LIN {X 0,Y 457.677,Z 380.613,A -85,B 0,C 180,E1 -16942.312,E2 -16942.312} C_VEL
LIN {X 0,Y 452.444,Z 370.143,A -85,B 0,C 180,E1 -16943.24,E2 -16943.24} C_VEL
LIN {X 0,Y 446.614,Z 360.173,A -85,B 0,C 180,E1 -16944.308,E2 -16944.308} C_VEL
LIN {X 0,Y 441.723,Z 352.476,A -85,B 0,C 180,E1 -16945.27,E2 -16945.27} C_VEL
LIN {X 0,Y 439.765,Z 349.442,A -85,B 0,C 180,E1 -16945.668,E2 -16945.668} C_VEL
LIN {X 0,Y 438.909,Z 348.163,A -85,B 0,C 180,E1 -16945.842,E2 -16945.842} C_VEL
LIN {X 0,Y 436.998,Z 345.517,A -85,B 0,C 180,E1 -16946.247,E2 -16946.247} C_VEL
LIN {X 0,Y 436.487,Z 343.674,A -85,B 0,C 180,E1 -16946.435,E2 -16946.435} C_VEL
LIN {X 0,Y 436.475,Z 343.673,A -85,B 0,C 180,E1 -16948.779,E2 -16948.779} C_VEL
LIN {X 0,Y 436.468,Z 343.672,A -85,B 0,C 180,E1 -16951.977,E2 -16951.977} C_VEL
LIN {X 0,Y 436.477,Z 343.666,A -85,B 0,C 180,E1 -16955.29,E2 -16955.29} C_VEL
LIN {X 0,Y 436.436,Z 343.668,A -85,B 0,C 180,E1 -16958.75,E2 -16958.75} C_VEL
LIN {X 0,Y 436.445,Z 343.67,A -85,B 0,C 180,E1 -16961.148,E2 -16961.148} C_VEL
LIN {X 0,Y 436.447,Z 343.671,A -85,B 0,C 180,E1 -16963.764,E2 -16963.764} C_VEL
LIN {X 0,Y 436.45,Z 343.673,A -85,B 0,C 180,E1 -16966.362,E2 -16966.362} C_VEL
LIN {X 0,Y 436.423,Z 343.682,A -85,B 0,C 180,E1 -16968.967,E2 -16968.967} C_VEL
LIN {X 0,Y 436.425,Z 343.682,A -85,B 0,C 180,E1 -16972.419,E2 -16972.419} C_VEL
LIN {X 0,Y 436.431,Z 343.811,A -85,B 0,C 180,E1 -16975.755,E2 -16975.755} C_VEL
LIN {X 0,Y 440.459,Z 359.383,A -85,B 0,C 180,E1 -16978.559,E2 -16978.559} C_VEL
LIN {X 0,Y 443.529,Z 373.428,A -85,B 0,C 180,E1 -16980.947,E2 -16980.947} C_VEL
LIN {X 0,Y 444.042,Z 376.825,A -85,B 0,C 180,E1 -16981.499,E2 -16981.499} C_VEL
LIN {X 0,Y 442.672,Z 390.65,A -85,B 0,C 180,E1 -16983.511,E2 -16983.511} C_VEL
LIN {X 0,Y 443.709,Z 396.754,A -85,B 0,C 180,E1 -16983.869,E2 -16983.869} C_VEL
LIN {X 0,Y 447.375,Z 420.193,A -85,B 0,C 180,E1 -16985.137,E2 -16985.137} C_VEL
LIN {X 0,Y 449.599,Z 437.106,A -85,B 0,C 180,E1 -16985.947,E2 -16985.947} C_VEL
LIN {X 0,Y 451.261,Z 453.177,A -85,B 0,C 180,E1 -16986.628,E2 -16986.628} C_VEL
LIN {X 0,Y 452.377,Z 476.599,A -85,B 0,C 180,E1 -16987.477,E2 -16987.477} C_VEL
LIN {X 0,Y 448.009,Z 553.44,A -85,B 0,C 180,E1 -16989.404,E2 -16989.404} C_VEL
LIN {X 0,Y 446.573,Z 569.624,A -85,B 0,C 180,E1 -16989.993,E2 -16989.993} C_VEL
LIN {X 0,Y 444.876,Z 583.938,A -85,B 0,C 180,E1 -16990.692,E2 -16990.692} C_VEL
LIN {X 0,Y 443.084,Z 597.736,A -85,B 0,C 180,E1 -16991.568,E2 -16991.568} C_VEL
LIN {X 0,Y 440.902,Z 615.075,A -85,B 0,C 180,E1 -16992.908,E2 -16992.908} C_VEL
LIN {X 0,Y 439.422,Z 626.686,A -85,B 0,C 180,E1 -16994.04,E2 -16994.04} C_VEL
LIN {X 0,Y 438.078,Z 636.36,A -85,B 0,C 180,E1 -16995.177,E2 -16995.177} C_VEL
LIN {X 0,Y 436.955,Z 646.109,A -85,B 0,C 180,E1 -16996.559,E2 -16996.559} C_VEL
LIN {X 0,Y 436.4,Z 651.742,A -85,B 0,C 180,E1 -16997.486,E2 -16997.486} C_VEL
LIN {X 0,Y 435.744,Z 662.573,A -85,B 0,C 180,E1 -16998.749,E2 -16998.749} C_VEL
LIN {X 0,Y 435.303,Z 671.76,A -85,B 0,C 180,E1 -17000.039,E2 -17000.039} C_VEL
LIN {X 0,Y 434.928,Z 680.021,A -85,B 0,C 180,E1 -17001.433,E2 -17001.433} C_VEL
LIN {X 0,Y 434.668,Z 687.893,A -85,B 0,C 180,E1 -17003.058,E2 -17003.058} C_VEL
LIN {X 0,Y 434.564,Z 693.312,A -85,B 0,C 180,E1 -17004.45,E2 -17004.45} C_VEL
LIN {X 0,Y 434.439,Z 697.641,A -85,B 0,C 180,E1 -17005.839,E2 -17005.839} C_VEL
LIN {X 0,Y 434.396,Z 701.016,A -85,B 0,C 180,E1 -17007.227,E2 -17007.227} C_VEL
LIN {X 0,Y 434.402,Z 703.511,A -85,B 0,C 180,E1 -17008.614,E2 -17008.614} C_VEL
LIN {X 0,Y 434.384,Z 705.081,A -85,B 0,C 180,E1 -17010,E2 -17010} C_VEL
LIN {X 0,Y 434.419,Z 705.916,A -85,B 0,C 180,E1 -17011.848,E2 -17011.848} C_VEL
LIN {X 0,Y 434.466,Z 705.265,A -85,B 0,C 180,E1 -17013.697,E2 -17013.697} C_VEL
LIN {X 0,Y 434.713,Z 703.119,A -85,B 0,C 180,E1 -17015.548,E2 -17015.548} C_VEL
LIN {X 0,Y 435.174,Z 699.48,A -85,B 0,C 180,E1 -17017.398,E2 -17017.398} C_VEL
LIN {X 0,Y 435.868,Z 694.257,A -85,B 0,C 180,E1 -17019.247,E2 -17019.247} C_VEL
LIN {X 0,Y 436.699,Z 689.192,A -85,B 0,C 180,E1 -17020.629,E2 -17020.629} C_VEL
LIN {X 0,Y 437.941,Z 681.532,A -85,B 0,C 180,E1 -17022.309,E2 -17022.309} C_VEL
LIN {X 0,Y 439.27,Z 672.935,A -85,B 0,C 180,E1 -17023.838,E2 -17023.838} C_VEL
LIN {X 0,Y 440.847,Z 663.536,A -85,B 0,C 180,E1 -17025.198,E2 -17025.198} C_VEL
LIN {X 0,Y 442.451,Z 652.225,A -85,B 0,C 180,E1 -17026.556,E2 -17026.556} C_VEL
LIN {X 0,Y 444.327,Z 639.573,A -85,B 0,C 180,E1 -17027.784,E2 -17027.784} C_VEL
LIN {X 0,Y 446.052,Z 626.94,A -85,B 0,C 180,E1 -17028.779,E2 -17028.779} C_VEL
LIN {X 0,Y 447.529,Z 613.948,A -85,B 0,C 180,E1 -17029.604,E2 -17029.604} C_VEL
LIN {X 0,Y 449.037,Z 599.167,A -85,B 0,C 180,E1 -17030.328,E2 -17030.328} C_VEL
LIN {X 0,Y 450.408,Z 583.991,A -85,B 0,C 180,E1 -17030.866,E2 -17030.866} C_VEL
LIN {X 0,Y 456.645,Z 487.44,A -85,B 0,C 180,E1 -17033.354,E2 -17033.354} C_VEL
LIN {X 0,Y 457.242,Z 476.209,A -85,B 0,C 180,E1 -17033.674,E2 -17033.674} C_VEL
LIN {X 0,Y 456.643,Z 460.353,A -85,B 0,C 180,E1 -17034.284,E2 -17034.284} C_VEL
LIN {X 0,Y 454.633,Z 438.662,A -85,B 0,C 180,E1 -17035.296,E2 -17035.296} C_VEL
LIN {X 0,Y 454.42,Z 436.088,A -85,B 0,C 180,E1 -17035.446,E2 -17035.446} C_VEL
LIN {X 0,Y 454.349,Z 415.095,A -85,B 0,C 180,E1 -17037.094,E2 -17037.094} C_VEL
LIN {X 0,Y 454.414,Z 399.172,A -85,B 0,C 180,E1 -17038.545,E2 -17038.545} C_VEL
LIN {X 0,Y 454.669,Z 389.171,A -85,B 0,C 180,E1 -17039.537,E2 -17039.537} C_VEL
LIN {X 0,Y 454.757,Z 385.084,A -85,B 0,C 180,E1 -17039.972,E2 -17039.972} C_VEL
LIN {X 0,Y 453.574,Z 375.492,A -85,B 0,C 180,E1 -17041.419,E2 -17041.419} C_VEL
LIN {X 0,Y 453.221,Z 371.903,A -85,B 0,C 180,E1 -17042.027,E2 -17042.027} C_VEL
LIN {X 0,Y 451.396,Z 368.316,A -85,B 0,C 180,E1 -17043.078,E2 -17043.078} C_VEL
LIN {X 0,Y 448.758,Z 363.877,A -85,B 0,C 180,E1 -17044.765,E2 -17044.765} C_VEL
LIN {X 0,Y 446.279,Z 359.984,A -85,B 0,C 180,E1 -17046.826,E2 -17046.826} C_VEL
LIN {X 0,Y 445.144,Z 358.305,A -85,B 0,C 180,E1 -17048.116,E2 -17048.116} C_VEL
LIN {X 0,Y 443.873,Z 356.858,A -85,B 0,C 180,E1 -17050.315,E2 -17050.315} C_VEL
LIN {X 0,Y 443.562,Z 356.547,A -85,B 0,C 180,E1 -17052.082,E2 -17052.082} C_VEL
LIN {X 0,Y 443.886,Z 357.081,A -85,B 0,C 180,E1 -17053.972,E2 -17053.972} C_VEL
LIN {X 0,Y 444.508,Z 357.779,A -85,B 0,C 180,E1 -17055.162,E2 -17055.162} C_VEL
LIN {X 0,Y 445.079,Z 359.312,A -85,B 0,C 180,E1 -17056.38,E2 -17056.38} C_VEL
LIN {X 0,Y 446.306,Z 361.926,A -85,B 0,C 180,E1 -17058.075,E2 -17058.075} C_VEL
LIN {X 0,Y 448.189,Z 366.353,A -85,B 0,C 180,E1 -17060.152,E2 -17060.152} C_VEL
LIN {X 0,Y 450.674,Z 372.66,A -85,B 0,C 180,E1 -17062.434,E2 -17062.434} C_VEL
LIN {X 0,Y 452.888,Z 379.057,A -85,B 0,C 180,E1 -17064.318,E2 -17064.318} C_VEL
LIN {X 0,Y 455.207,Z 387.381,A -85,B 0,C 180,E1 -17066.362,E2 -17066.362} C_VEL
LIN {X 0,Y 457.231,Z 396.879,A -85,B 0,C 180,E1 -17068.361,E2 -17068.361} C_VEL
LIN {X 0,Y 457.648,Z 400.955,A -85,B 0,C 180,E1 -17069.093,E2 -17069.093} C_VEL
LIN {X 0,Y 454.383,Z 422.257,A -85,B 0,C 180,E1 -17072.001,E2 -17072.001} C_VEL
LIN {X 0,Y 451.946,Z 440.08,A -85,B 0,C 180,E1 -17074.351,E2 -17074.351} C_VEL
LIN {X 0,Y 455.098,Z 456.713,A -85,B 0,C 180,E1 -17075.326,E2 -17075.326} C_VEL
LIN {X 0,Y 457.268,Z 472.318,A -85,B 0,C 180,E1 -17076.103,E2 -17076.103} C_VEL
LIN {X 0,Y 457.699,Z 477.669,A -85,B 0,C 180,E1 -17076.329,E2 -17076.329} C_VEL
LIN {X 0,Y 452.325,Z 559.762,A -85,B 0,C 180,E1 -17078.428,E2 -17078.428} C_VEL
LIN {X 0,Y 450.776,Z 583.934,A -85,B 0,C 180,E1 -17079.06,E2 -17079.06} C_VEL
LIN {X 0,Y 449.354,Z 599.265,A -85,B 0,C 180,E1 -17079.647,E2 -17079.647} C_VEL
LIN {X 0,Y 447.901,Z 613.022,A -85,B 0,C 180,E1 -17080.353,E2 -17080.353} C_VEL
LIN {X 0,Y 446.285,Z 626.426,A -85,B 0,C 180,E1 -17081.232,E2 -17081.232} C_VEL
LIN {X 0,Y 444.402,Z 639.894,A -85,B 0,C 180,E1 -17082.338,E2 -17082.338} C_VEL
LIN {X 0,Y 442.623,Z 652.052,A -85,B 0,C 180,E1 -17083.569,E2 -17083.569} C_VEL
LIN {X 0,Y 440.999,Z 662.166,A -85,B 0,C 180,E1 -17084.807,E2 -17084.807} C_VEL
LIN {X 0,Y 439.496,Z 671.417,A -85,B 0,C 180,E1 -17086.169,E2 -17086.169} C_VEL
LIN {X 0,Y 438.119,Z 680.312,A -85,B 0,C 180,E1 -17087.782,E2 -17087.782} C_VEL
LIN {X 0,Y 436.881,Z 687.469,A -85,B 0,C 180,E1 -17089.375,E2 -17089.375} C_VEL
LIN {X 0,Y 436.048,Z 692.49,A -85,B 0,C 180,E1 -17090.756,E2 -17090.756} C_VEL
LIN {X 0,Y 435.249,Z 697.663,A -85,B 0,C 180,E1 -17092.603,E2 -17092.603} C_VEL
LIN {X 0,Y 434.706,Z 701.272,A -85,B 0,C 180,E1 -17094.452,E2 -17094.452} C_VEL
LIN {X 0,Y 434.444,Z 703.403,A -85,B 0,C 180,E1 -17096.303,E2 -17096.303} C_VEL
LIN {X 0,Y 434.35,Z 704.067,A -85,B 0,C 180,E1 -17098.152,E2 -17098.152} C_VEL
LIN {X 0,Y 434.316,Z 703.251,A -85,B 0,C 180,E1 -17100,E2 -17100} C_VEL
LIN {X 0,Y 434.35,Z 700.967,A -85,B 0,C 180,E1 -17101.849,E2 -17101.849} C_VEL
LIN {X 0,Y 434.349,Z 698.27,A -85,B 0,C 180,E1 -17103.236,E2 -17103.236} C_VEL
LIN {X 0,Y 434.441,Z 694.648,A -85,B 0,C 180,E1 -17104.624,E2 -17104.624} C_VEL
LIN {X 0,Y 434.575,Z 689.804,A -85,B 0,C 180,E1 -17106.07,E2 -17106.07} C_VEL
LIN {X 0,Y 434.826,Z 683.278,A -85,B 0,C 180,E1 -17107.637,E2 -17107.637} C_VEL
LIN {X 0,Y 435.223,Z 674.843,A -85,B 0,C 180,E1 -17109.262,E2 -17109.262} C_VEL
LIN {X 0,Y 435.755,Z 665.995,A -85,B 0,C 180,E1 -17110.653,E2 -17110.653} C_VEL
LIN {X 0,Y 436.232,Z 656.984,A -85,B 0,C 180,E1 -17111.843,E2 -17111.843} C_VEL
LIN {X 0,Y 436.876,Z 645.666,A -85,B 0,C 180,E1 -17113.089,E2 -17113.089} C_VEL
LIN {X 0,Y 437.653,Z 632.877,A -85,B 0,C 180,E1 -17114.245,E2 -17114.245} C_VEL
LIN {X 0,Y 438.37,Z 620.317,A -85,B 0,C 180,E1 -17115.168,E2 -17115.168} C_VEL
LIN {X 0,Y 439.097,Z 606.466,A -85,B 0,C 180,E1 -17115.973,E2 -17115.973} C_VEL
LIN {X 0,Y 439.608,Z 592.172,A -85,B 0,C 180,E1 -17116.607,E2 -17116.607} C_VEL
LIN {X 0,Y 440.169,Z 576.613,A -85,B 0,C 180,E1 -17117.094,E2 -17117.094} C_VEL
LIN {X 0,Y 442.754,Z 469.934,A -85,B 0,C 180,E1 -17119.451,E2 -17119.451} C_VEL
LIN {X 0,Y 439.834,Z 439.603,A -85,B 0,C 180,E1 -17120.233,E2 -17120.233} C_VEL
LIN {X 0,Y 441.544,Z 410.298,A -85,B 0,C 180,E1 -17123.861,E2 -17123.861} C_VEL
LIN {X 0,Y 443.123,Z 384.772,A -85,B 0,C 180,E1 -17127.03,E2 -17127.03} C_VEL
LIN {X 0,Y 443.661,Z 375.927,A -85,B 0,C 180,E1 -17128.132,E2 -17128.132} C_VEL
LIN {X 0,Y 439.991,Z 358.902,A -85,B 0,C 180,E1 -17130.454,E2 -17130.454} C_VEL
LIN {X 0,Y 436.523,Z 343.668,A -85,B 0,C 180,E1 -17132.584,E2 -17132.584} C_VEL
LIN {X 0,Y 436.491,Z 343.675,A -85,B 0,C 180,E1 -17135.289,E2 -17135.289} C_VEL
LIN {X 0,Y 436.468,Z 343.673,A -85,B 0,C 180,E1 -17138.747,E2 -17138.747} C_VEL
LIN {X 0,Y 436.48,Z 343.675,A -85,B 0,C 180,E1 -17141.144,E2 -17141.144} C_VEL
LIN {X 0,Y 436.472,Z 343.67,A -85,B 0,C 180,E1 -17143.767,E2 -17143.767} C_VEL
LIN {X 0,Y 436.472,Z 343.671,A -85,B 0,C 180,E1 -17146.365,E2 -17146.365} C_VEL
LIN {X 0,Y 436.483,Z 343.674,A -85,B 0,C 180,E1 -17148.959,E2 -17148.959} C_VEL
LIN {X 0,Y 436.459,Z 343.675,A -85,B 0,C 180,E1 -17152.422,E2 -17152.422} C_VEL
LIN {X 0,Y 436.479,Z 343.669,A -85,B 0,C 180,E1 -17155.829,E2 -17155.829} C_VEL
LIN {X 0,Y 436.467,Z 343.671,A -85,B 0,C 180,E1 -17159.1,E2 -17159.1} C_VEL
LIN {X 0,Y 436.5,Z 343.672,A -85,B 0,C 180,E1 -17162.267,E2 -17162.267} C_VEL
LIN {X 0,Y 436.453,Z 343.672,A -85,B 0,C 180,E1 -17165.338,E2 -17165.338} C_VEL
LIN {X 0,Y 436.49,Z 343.674,A -85,B 0,C 180,E1 -17168.341,E2 -17168.341} C_VEL
LIN {X 0,Y 436.536,Z 343.663,A -85,B 0,C 180,E1 -17171.282,E2 -17171.282} C_VEL
LIN {X 0,Y 436.539,Z 343.669,A -85,B 0,C 180,E1 -17173.973,E2 -17173.973} C_VEL
LIN {X 0,Y 438.742,Z 349.624,A -85,B 0,C 180,E1 -17174.188,E2 -17174.188} C_VEL
LIN {X 0,Y 445.557,Z 367.49,A -85,B 0,C 180,E1 -17174.799,E2 -17174.799} C_VEL
LIN {X 0,Y 444.443,Z 456.819,A -85,B 0,C 180,E1 -17176.24,E2 -17176.24} C_VEL
LIN {X 0,Y 444.336,Z 471.415,A -85,B 0,C 180,E1 -17176.584,E2 -17176.584} C_VEL
LIN {X 0,Y 443.999,Z 484.727,A -85,B 0,C 180,E1 -17177.067,E2 -17177.067} C_VEL
LIN {X 0,Y 443.418,Z 497.369,A -85,B 0,C 180,E1 -17177.687,E2 -17177.687} C_VEL
LIN {X 0,Y 442.709,Z 509.826,A -85,B 0,C 180,E1 -17178.478,E2 -17178.478} C_VEL
LIN {X 0,Y 441.998,Z 522.081,A -85,B 0,C 180,E1 -17179.46,E2 -17179.46} C_VEL
LIN {X 0,Y 440.993,Z 533.977,A -85,B 0,C 180,E1 -17180.63,E2 -17180.63} C_VEL
LIN {X 0,Y 440.059,Z 543.484,A -85,B 0,C 180,E1 -17181.764,E2 -17181.764} C_VEL
LIN {X 0,Y 439.03,Z 553.01,A -85,B 0,C 180,E1 -17183.128,E2 -17183.128} C_VEL
LIN {X 0,Y 438.195,Z 560.908,A -85,B 0,C 180,E1 -17184.497,E2 -17184.497} C_VEL
LIN {X 0,Y 437.468,Z 567.499,A -85,B 0,C 180,E1 -17185.868,E2 -17185.868} C_VEL
LIN {X 0,Y 436.897,Z 572.99,A -85,B 0,C 180,E1 -17187.243,E2 -17187.243} C_VEL
LIN {X 0,Y 436.368,Z 578.741,A -85,B 0,C 180,E1 -17189.08,E2 -17189.08} C_VEL
LIN {X 0,Y 436.014,Z 582.966,A -85,B 0,C 180,E1 -17190.921,E2 -17190.921} C_VEL
LIN {X 0,Y 435.921,Z 585.784,A -85,B 0,C 180,E1 -17192.763,E2 -17192.763} C_VEL
LIN {X 0,Y 435.817,Z 587.301,A -85,B 0,C 180,E1 -17194.609,E2 -17194.609} C_VEL
LIN {X 0,Y 436.001,Z 587.512,A -85,B 0,C 180,E1 -17196.457,E2 -17196.457} C_VEL
LIN {X 0,Y 436.222,Z 586.445,A -85,B 0,C 180,E1 -17198.309,E2 -17198.309} C_VEL
LIN {X 0,Y 436.612,Z 584.058,A -85,B 0,C 180,E1 -17200.164,E2 -17200.164} C_VEL
LIN {X 0,Y 437.413,Z 580.231,A -85,B 0,C 180,E1 -17202.016,E2 -17202.016} C_VEL
LIN {X 0,Y 438.269,Z 574.861,A -85,B 0,C 180,E1 -17203.871,E2 -17203.871} C_VEL
LIN {X 0,Y 439.123,Z 569.75,A -85,B 0,C 180,E1 -17205.26,E2 -17205.26} C_VEL
LIN {X 0,Y 440.079,Z 563.506,A -85,B 0,C 180,E1 -17206.648,E2 -17206.648} C_VEL
LIN {X 0,Y 440.565,Z 560.276,A -85,B 0,C 180,E1 -17207.273,E2 -17207.273} C_VEL
LIN {X 0,Y 440.422,Z 556.973,A -85,B 0,C 180,E1 -17207.912,E2 -17207.912} C_VEL
LIN {X 0,Y 438.511,Z 551.47,A -85,B 0,C 180,E1 -17208.962,E2 -17208.962} C_VEL
LIN {X 0,Y 436.643,Z 545.441,A -85,B 0,C 180,E1 -17209.963,E2 -17209.963} C_VEL
LIN {X 0,Y 436.555,Z 541.317,A -85,B 0,C 180,E1 -17210.517,E2 -17210.517} C_VEL
LIN {X 0,Y 437.884,Z 530.282,A -85,B 0,C 180,E1 -17211.755,E2 -17211.755} C_VEL
LIN {X 0,Y 439.035,Z 519.376,A -85,B 0,C 180,E1 -17212.761,E2 -17212.761} C_VEL
LIN {X 0,Y 440.224,Z 506.915,A -85,B 0,C 180,E1 -17213.688,E2 -17213.688} C_VEL
LIN {X 0,Y 440.86,Z 495.16,A -85,B 0,C 180,E1 -17214.399,E2 -17214.399} C_VEL
LIN {X 0,Y 441.544,Z 480.938,A -85,B 0,C 180,E1 -17215.046,E2 -17215.046} C_VEL
LIN {X 0,Y 441.906,Z 467.059,A -85,B 0,C 180,E1 -17215.486,E2 -17215.486} C_VEL
LIN {X 0,Y 442.223,Z 442.075,A -85,B 0,C 180,E1 -17215.945,E2 -17215.945} C_VEL
LIN {X 0,Y 443.528,Z 375.813,A -85,B 0,C 180,E1 -17217.024,E2 -17217.024} C_VEL
LIN {X 0,Y 433.277,Z 353.124,A -85,B 0,C 180,E1 -17218.061,E2 -17218.061} C_VEL
LIN {X 0,Y 429.628,Z 345.62,A -85,B 0,C 180,E1 -17218.434,E2 -17218.434} C_VEL
LIN {X 0,Y 429.415,Z 344.551,A -85,B 0,C 180,E1 -17218.479,E2 -17218.479} C_VEL
LIN {X 0,Y 429.376,Z 344.556,A -85,B 0,C 180,E1 -17221.468,E2 -17221.468} C_VEL
LIN {X 0,Y 429.34,Z 344.563,A -85,B 0,C 180,E1 -17224.821,E2 -17224.821} C_VEL
LIN {X 0,Y 429.386,Z 344.556,A -85,B 0,C 180,E1 -17227.126,E2 -17227.126} C_VEL
LIN {X 0,Y 429.37,Z 344.561,A -85,B 0,C 180,E1 -17230.733,E2 -17230.733} C_VEL
LIN {X 0,Y 429.394,Z 344.557,A -85,B 0,C 180,E1 -17234.131,E2 -17234.131} C_VEL
LIN {X 0,Y 429.383,Z 344.556,A -85,B 0,C 180,E1 -17237.23,E2 -17237.23} C_VEL
LIN {X 0,Y 429.369,Z 344.553,A -85,B 0,C 180,E1 -17240.489,E2 -17240.489} C_VEL
LIN {X 0,Y 429.383,Z 344.521,A -85,B 0,C 180,E1 -17243.066,E2 -17243.066} C_VEL
LIN {X 0,Y 429.393,Z 344.553,A -85,B 0,C 180,E1 -17246.315,E2 -17246.315} C_VEL
LIN {X 0,Y 429.408,Z 344.545,A -85,B 0,C 180,E1 -17249.83,E2 -17249.83} C_VEL
LIN {X 0,Y 429.427,Z 344.546,A -85,B 0,C 180,E1 -17252.824,E2 -17252.824} C_VEL
LIN {X 0,Y 429.42,Z 344.554,A -85,B 0,C 180,E1 -17255.986,E2 -17255.986} C_VEL
LIN {X 0,Y 429.446,Z 344.543,A -85,B 0,C 180,E1 -17259.386,E2 -17259.386} C_VEL
LIN {X 0,Y 435.371,Z 365.507,A -85,B 0,C 180,E1 -17260.041,E2 -17260.041} C_VEL
LIN {X 0,Y 433.262,Z 463.185,A -85,B 0,C 180,E1 -17262.23,E2 -17262.23} C_VEL
LIN {X 0,Y 433.081,Z 478.715,A -85,B 0,C 180,E1 -17262.783,E2 -17262.783} C_VEL
LIN {X 0,Y 432.555,Z 492.998,A -85,B 0,C 180,E1 -17263.477,E2 -17263.477} C_VEL
LIN {X 0,Y 432.049,Z 506.957,A -85,B 0,C 180,E1 -17264.364,E2 -17264.364} C_VEL
LIN {X 0,Y 431.479,Z 518.961,A -85,B 0,C 180,E1 -17265.306,E2 -17265.306} C_VEL
LIN {X 0,Y 430.809,Z 531.324,A -85,B 0,C 180,E1 -17266.483,E2 -17266.483} C_VEL
LIN {X 0,Y 430.388,Z 542.523,A -85,B 0,C 180,E1 -17267.785,E2 -17267.785} C_VEL
LIN {X 0,Y 429.822,Z 552.611,A -85,B 0,C 180,E1 -17269.198,E2 -17269.198} C_VEL
LIN {X 0,Y 429.319,Z 561.019,A -85,B 0,C 180,E1 -17270.61,E2 -17270.61} C_VEL
LIN {X 0,Y 428.966,Z 569.102,A -85,B 0,C 180,E1 -17272.258,E2 -17272.258} C_VEL
LIN {X 0,Y 428.738,Z 575.578,A -85,B 0,C 180,E1 -17273.904,E2 -17273.904} C_VEL
LIN {X 0,Y 428.671,Z 580.161,A -85,B 0,C 180,E1 -17275.372,E2 -17275.372} C_VEL
LIN {X 0,Y 428.671,Z 584.435,A -85,B 0,C 180,E1 -17277.19,E2 -17277.19} C_VEL
LIN {X 0,Y 428.814,Z 587.335,A -85,B 0,C 180,E1 -17279.064,E2 -17279.064} C_VEL
LIN {X 0,Y 429.067,Z 588.81,A -85,B 0,C 180,E1 -17280.935,E2 -17280.935} C_VEL
LIN {X 0,Y 429.536,Z 588.855,A -85,B 0,C 180,E1 -17282.804,E2 -17282.804} C_VEL
LIN {X 0,Y 430.323,Z 587.416,A -85,B 0,C 180,E1 -17284.668,E2 -17284.668} C_VEL
LIN {X 0,Y 431.215,Z 584.507,A -85,B 0,C 180,E1 -17286.529,E2 -17286.529} C_VEL
LIN {X 0,Y 432.085,Z 581.348,A -85,B 0,C 180,E1 -17287.92,E2 -17287.92} C_VEL
LIN {X 0,Y 433.676,Z 575.565,A -85,B 0,C 180,E1 -17289.764,E2 -17289.764} C_VEL
LIN {X 0,Y 435.028,Z 569.083,A -85,B 0,C 180,E1 -17291.375,E2 -17291.375} C_VEL
LIN {X 0,Y 436.68,Z 560.948,A -85,B 0,C 180,E1 -17292.977,E2 -17292.977} C_VEL
LIN {X 0,Y 438.219,Z 552.383,A -85,B 0,C 180,E1 -17294.344,E2 -17294.344} C_VEL
LIN {X 0,Y 439.852,Z 542.059,A -85,B 0,C 180,E1 -17295.707,E2 -17295.707} C_VEL
LIN {X 0,Y 441.593,Z 530.502,A -85,B 0,C 180,E1 -17296.945,E2 -17296.945} C_VEL
LIN {X 0,Y 443.229,Z 518.188,A -85,B 0,C 180,E1 -17298.015,E2 -17298.015} C_VEL
LIN {X 0,Y 444.645,Z 504.392,A -85,B 0,C 180,E1 -17298.982,E2 -17298.982} C_VEL
LIN {X 0,Y 445.684,Z 490.634,A -85,B 0,C 180,E1 -17299.749,E2 -17299.749} C_VEL
LIN {X 0,Y 446.485,Z 476.415,A -85,B 0,C 180,E1 -17300.34,E2 -17300.34} C_VEL
LIN {X 0,Y 447.172,Z 458.257,A -85,B 0,C 180,E1 -17300.876,E2 -17300.876} C_VEL
LIN {X 0,Y 452.155,Z 383.344,A -85,B 0,C 180,E1 -17302.816,E2 -17302.816} C_VEL
LIN {X 0,Y 446.936,Z 372.943,A -85,B 0,C 180,E1 -17303.795,E2 -17303.795} C_VEL
LIN {X 0,Y 441.418,Z 363.583,A -85,B 0,C 180,E1 -17304.862,E2 -17304.862} C_VEL
LIN {X 0,Y 437.481,Z 357.481,A -85,B 0,C 180,E1 -17305.66,E2 -17305.66} C_VEL
LIN {X 0,Y 434.973,Z 353.534,A -85,B 0,C 180,E1 -17306.205,E2 -17306.205} C_VEL
LIN {X 0,Y 432.902,Z 350.308,A -85,B 0,C 180,E1 -17306.683,E2 -17306.683} C_VEL
LIN {X 0,Y 432.416,Z 349.473,A -85,B 0,C 180,E1 -17306.8,E2 -17306.8} C_VEL
LIN {X 0,Y 430.428,Z 347.394,A -85,B 0,C 180,E1 -17307.222,E2 -17307.222} C_VEL
LIN {X 0,Y 429.475,Z 344.803,A -85,B 0,C 180,E1 -17307.501,E2 -17307.501} C_VEL
LIN {X 0,Y 429.461,Z 344.548,A -85,B 0,C 180,E1 -17307.567,E2 -17307.567} C_VEL
LIN {X 0,Y 429.418,Z 344.551,A -85,B 0,C 180,E1 -17310.375,E2 -17310.375} C_VEL
LIN {X 0,Y 429.433,Z 344.546,A -85,B 0,C 180,E1 -17313.709,E2 -17313.709} C_VEL
LIN {X 0,Y 429.409,Z 344.544,A -85,B 0,C 180,E1 -17317.123,E2 -17317.123} C_VEL
LIN {X 0,Y 429.415,Z 344.545,A -85,B 0,C 180,E1 -17319.946,E2 -17319.946} C_VEL
LIN {X 0,Y 429.378,Z 344.556,A -85,B 0,C 180,E1 -17323.247,E2 -17323.247} C_VEL
LIN {X 0,Y 429.401,Z 344.55,A -85,B 0,C 180,E1 -17325.868,E2 -17325.868} C_VEL
LIN {X 0,Y 429.37,Z 344.558,A -85,B 0,C 180,E1 -17329.267,E2 -17329.267} C_VEL
LIN {X 0,Y 429.381,Z 344.557,A -85,B 0,C 180,E1 -17332.873,E2 -17332.873} C_VEL
LIN {X 0,Y 429.395,Z 344.592,A -85,B 0,C 180,E1 -17335.346,E2 -17335.346} C_VEL
LIN {X 0,Y 433.558,Z 360.83,A -85,B 0,C 180,E1 -17338.328,E2 -17338.328} C_VEL
LIN {X 0,Y 436.89,Z 376.234,A -85,B 0,C 180,E1 -17340.988,E2 -17340.988} C_VEL
LIN {X 0,Y 437.103,Z 380.303,A -85,B 0,C 180,E1 -17341.637,E2 -17341.637} C_VEL
LIN {X 0,Y 436.435,Z 386.351,A -85,B 0,C 180,E1 -17342.522,E2 -17342.522} C_VEL
LIN {X 0,Y 437.356,Z 392.245,A -85,B 0,C 180,E1 -17342.875,E2 -17342.875} C_VEL
LIN {X 0,Y 439.054,Z 402.862,A -85,B 0,C 180,E1 -17343.522,E2 -17343.522} C_VEL
LIN {X 0,Y 441.76,Z 420.595,A -85,B 0,C 180,E1 -17344.514,E2 -17344.514} C_VEL
LIN {X 0,Y 443.998,Z 437.926,A -85,B 0,C 180,E1 -17345.379,E2 -17345.379} C_VEL
LIN {X 0,Y 445.575,Z 454.469,A -85,B 0,C 180,E1 -17346.115,E2 -17346.115} C_VEL
LIN {X 0,Y 446.578,Z 477.848,A -85,B 0,C 180,E1 -17346.974,E2 -17346.974} C_VEL
LIN {X 0,Y 441.948,Z 553.39,A -85,B 0,C 180,E1 -17348.926,E2 -17348.926} C_VEL
LIN {X 0,Y 440.444,Z 569.224,A -85,B 0,C 180,E1 -17349.52,E2 -17349.52} C_VEL
LIN {X 0,Y 438.553,Z 584.129,A -85,B 0,C 180,E1 -17350.281,E2 -17350.281} C_VEL
LIN {X 0,Y 436.631,Z 597.911,A -85,B 0,C 180,E1 -17351.188,E2 -17351.188} C_VEL
LIN {X 0,Y 434.645,Z 611.385,A -85,B 0,C 180,E1 -17352.291,E2 -17352.291} C_VEL
LIN {X 0,Y 432.424,Z 627.285,A -85,B 0,C 180,E1 -17353.895,E2 -17353.895} C_VEL
LIN {X 0,Y 430.944,Z 637.619,A -85,B 0,C 180,E1 -17355.167,E2 -17355.167} C_VEL
LIN {X 0,Y 429.85,Z 647.024,A -85,B 0,C 180,E1 -17356.573,E2 -17356.573} C_VEL
LIN {X 0,Y 429.272,Z 652.853,A -85,B 0,C 180,E1 -17357.574,E2 -17357.574} C_VEL
LIN {X 0,Y 428.553,Z 663.612,A -85,B 0,C 180,E1 -17358.872,E2 -17358.872} C_VEL
LIN {X 0,Y 428.182,Z 672.15,A -85,B 0,C 180,E1 -17360.109,E2 -17360.109} C_VEL
LIN {X 0,Y 427.808,Z 680.356,A -85,B 0,C 180,E1 -17361.526,E2 -17361.526} C_VEL
LIN {X 0,Y 427.603,Z 687.136,A -85,B 0,C 180,E1 -17362.943,E2 -17362.943} C_VEL
LIN {X 0,Y 427.475,Z 692.692,A -85,B 0,C 180,E1 -17364.358,E2 -17364.358} C_VEL
LIN {X 0,Y 427.364,Z 697.161,A -85,B 0,C 180,E1 -17365.77,E2 -17365.77} C_VEL
LIN {X 0,Y 427.32,Z 700.663,A -85,B 0,C 180,E1 -17367.181,E2 -17367.181} C_VEL
LIN {X 0,Y 427.347,Z 702.464,A -85,B 0,C 180,E1 -17368.121,E2 -17368.121} C_VEL
LIN {X 0,Y 427.31,Z 704.911,A -85,B 0,C 180,E1 -17370,E2 -17370} C_VEL
LIN {X 0,Y 427.319,Z 705.869,A -85,B 0,C 180,E1 -17371.879,E2 -17371.879} C_VEL
LIN {X 0,Y 427.375,Z 705.354,A -85,B 0,C 180,E1 -17373.759,E2 -17373.759} C_VEL
LIN {X 0,Y 427.644,Z 703.373,A -85,B 0,C 180,E1 -17375.64,E2 -17375.64} C_VEL
LIN {X 0,Y 428.13,Z 699.868,A -85,B 0,C 180,E1 -17377.521,E2 -17377.521} C_VEL
LIN {X 0,Y 428.872,Z 694.789,A -85,B 0,C 180,E1 -17379.4,E2 -17379.4} C_VEL
LIN {X 0,Y 429.771,Z 689.861,A -85,B 0,C 180,E1 -17380.803,E2 -17380.803} C_VEL
LIN {X 0,Y 431.049,Z 682.483,A -85,B 0,C 180,E1 -17382.49,E2 -17382.49} C_VEL
LIN {X 0,Y 432.468,Z 673.964,A -85,B 0,C 180,E1 -17384.06,E2 -17384.06} C_VEL
LIN {X 0,Y 434.123,Z 664.822,A -85,B 0,C 180,E1 -17385.44,E2 -17385.44} C_VEL
LIN {X 0,Y 435.806,Z 653.857,A -85,B 0,C 180,E1 -17386.816,E2 -17386.816} C_VEL
LIN {X 0,Y 437.736,Z 641.592,A -85,B 0,C 180,E1 -17388.061,E2 -17388.061} C_VEL
LIN {X 0,Y 439.738,Z 627.906,A -85,B 0,C 180,E1 -17389.179,E2 -17389.179} C_VEL
LIN {X 0,Y 441.438,Z 614.33,A -85,B 0,C 180,E1 -17390.068,E2 -17390.068} C_VEL
LIN {X 0,Y 443.096,Z 599.037,A -85,B 0,C 180,E1 -17390.832,E2 -17390.832} C_VEL
LIN {X 0,Y 444.553,Z 583.395,A -85,B 0,C 180,E1 -17391.391,E2 -17391.391} C_VEL
LIN {X 0,Y 451.193,Z 487.107,A -85,B 0,C 180,E1 -17393.938,E2 -17393.938} C_VEL
LIN {X 0,Y 451.757,Z 476.696,A -85,B 0,C 180,E1 -17394.246,E2 -17394.246} C_VEL
LIN {X 0,Y 451.19,Z 460.696,A -85,B 0,C 180,E1 -17394.889,E2 -17394.889} C_VEL
LIN {X 0,Y 449.324,Z 439.334,A -85,B 0,C 180,E1 -17395.926,E2 -17395.926} C_VEL
LIN {X 0,Y 449.036,Z 435.461,A -85,B 0,C 180,E1 -17396.175,E2 -17396.175} C_VEL
LIN {X 0,Y 449.273,Z 416.078,A -85,B 0,C 180,E1 -17397.76,E2 -17397.76} C_VEL
LIN {X 0,Y 449.507,Z 402.261,A -85,B 0,C 180,E1 -17399.064,E2 -17399.064} C_VEL
LIN {X 0,Y 450.009,Z 390.651,A -85,B 0,C 180,E1 -17400.253,E2 -17400.253} C_VEL
LIN {X 0,Y 449.98,Z 387.365,A -85,B 0,C 180,E1 -17400.669,E2 -17400.669} C_VEL
LIN {X 0,Y 449.064,Z 378.847,A -85,B 0,C 180,E1 -17402.028,E2 -17402.028} C_VEL
LIN {X 0,Y 448.599,Z 376.293,A -85,B 0,C 180,E1 -17402.525,E2 -17402.525} C_VEL
LIN {X 0,Y 446.45,Z 372.718,A -85,B 0,C 180,E1 -17403.744,E2 -17403.744} C_VEL
LIN {X 0,Y 444.665,Z 369.479,A -85,B 0,C 180,E1 -17405.004,E2 -17405.004} C_VEL
LIN {X 0,Y 442.362,Z 365.782,A -85,B 0,C 180,E1 -17406.992,E2 -17406.992} C_VEL
LIN {X 0,Y 440.791,Z 363.707,A -85,B 0,C 180,E1 -17408.864,E2 -17408.864} C_VEL
LIN {X 0,Y 439.84,Z 362.622,A -85,B 0,C 180,E1 -17410.762,E2 -17410.762} C_VEL
LIN {X 0,Y 439.701,Z 362.637,A -85,B 0,C 180,E1 -17413.235,E2 -17413.235} C_VEL
LIN {X 0,Y 440.062,Z 363.152,A -85,B 0,C 180,E1 -17414.455,E2 -17414.455} C_VEL
LIN {X 0,Y 440.568,Z 364.171,A -85,B 0,C 180,E1 -17415.679,E2 -17415.679} C_VEL
LIN {X 0,Y 442.14,Z 368.011,A -85,B 0,C 180,E1 -17418.289,E2 -17418.289} C_VEL
LIN {X 0,Y 444.09,Z 373.072,A -85,B 0,C 180,E1 -17420.611,E2 -17420.611} C_VEL
LIN {X 0,Y 446.367,Z 379.256,A -85,B 0,C 180,E1 -17422.801,E2 -17422.801} C_VEL
LIN {X 0,Y 448.409,Z 385.822,A -85,B 0,C 180,E1 -17424.693,E2 -17424.693} C_VEL
LIN {X 0,Y 450.392,Z 394.099,A -85,B 0,C 180,E1 -17426.683,E2 -17426.683} C_VEL
LIN {X 0,Y 451.938,Z 402.722,A -85,B 0,C 180,E1 -17428.477,E2 -17428.477} C_VEL
LIN {X 0,Y 451.798,Z 405.556,A -85,B 0,C 180,E1 -17428.939,E2 -17428.939} C_VEL
LIN {X 0,Y 448.067,Z 428.007,A -85,B 0,C 180,E1 -17432.032,E2 -17432.032} C_VEL
LIN {X 0,Y 446.412,Z 440.131,A -85,B 0,C 180,E1 -17433.645,E2 -17433.645} C_VEL
LIN {X 0,Y 449.67,Z 458.131,A -85,B 0,C 180,E1 -17434.747,E2 -17434.747} C_VEL
LIN {X 0,Y 451.796,Z 473.687,A -85,B 0,C 180,E1 -17435.557,E2 -17435.557} C_VEL
LIN {X 0,Y 452.193,Z 478.777,A -85,B 0,C 180,E1 -17435.782,E2 -17435.782} C_VEL
LIN {X 0,Y 446.365,Z 562.73,A -85,B 0,C 180,E1 -17437.982,E2 -17437.982} C_VEL
LIN {X 0,Y 444.798,Z 584.845,A -85,B 0,C 180,E1 -17438.585,E2 -17438.585} C_VEL
LIN {X 0,Y 443.319,Z 599.869,A -85,B 0,C 180,E1 -17439.176,E2 -17439.176} C_VEL
LIN {X 0,Y 441.684,Z 614.35,A -85,B 0,C 180,E1 -17439.944,E2 -17439.944} C_VEL
LIN {X 0,Y 439.762,Z 628.815,A -85,B 0,C 180,E1 -17440.943,E2 -17440.943} C_VEL
LIN {X 0,Y 437.838,Z 641.874,A -85,B 0,C 180,E1 -17442.064,E2 -17442.064} C_VEL
LIN {X 0,Y 436.134,Z 652.656,A -85,B 0,C 180,E1 -17443.197,E2 -17443.197} C_VEL
LIN {X 0,Y 434.274,Z 663.471,A -85,B 0,C 180,E1 -17444.566,E2 -17444.566} C_VEL
LIN {X 0,Y 432.697,Z 672.468,A -85,B 0,C 180,E1 -17445.947,E2 -17445.947} C_VEL
LIN {X 0,Y 431.233,Z 681.23,A -85,B 0,C 180,E1 -17447.592,E2 -17447.592} C_VEL
LIN {X 0,Y 429.938,Z 688.173,A -85,B 0,C 180,E1 -17449.202,E2 -17449.202} C_VEL
LIN {X 0,Y 429.055,Z 693.051,A -85,B 0,C 180,E1 -17450.604,E2 -17450.604} C_VEL
LIN {X 0,Y 428.207,Z 698.086,A -85,B 0,C 180,E1 -17452.481,E2 -17452.481} C_VEL
LIN {X 0,Y 427.638,Z 701.565,A -85,B 0,C 180,E1 -17454.36,E2 -17454.36} C_VEL
LIN {X 0,Y 427.358,Z 703.54,A -85,B 0,C 180,E1 -17456.241,E2 -17456.241} C_VEL
LIN {X 0,Y 427.262,Z 704.055,A -85,B 0,C 180,E1 -17458.121,E2 -17458.121} C_VEL
LIN {X 0,Y 427.233,Z 703.117,A -85,B 0,C 180,E1 -17460,E2 -17460} C_VEL
LIN {X 0,Y 427.262,Z 700.709,A -85,B 0,C 180,E1 -17461.879,E2 -17461.879} C_VEL
LIN {X 0,Y 427.297,Z 696.771,A -85,B 0,C 180,E1 -17463.76,E2 -17463.76} C_VEL
LIN {X 0,Y 427.385,Z 692.686,A -85,B 0,C 180,E1 -17465.172,E2 -17465.172} C_VEL
LIN {X 0,Y 427.548,Z 687.588,A -85,B 0,C 180,E1 -17466.585,E2 -17466.585} C_VEL
LIN {X 0,Y 427.831,Z 680.202,A -85,B 0,C 180,E1 -17468.237,E2 -17468.237} C_VEL
LIN {X 0,Y 428.265,Z 672.446,A -85,B 0,C 180,E1 -17469.651,E2 -17469.651} C_VEL
LIN {X 0,Y 428.727,Z 663.103,A -85,B 0,C 180,E1 -17471.068,E2 -17471.068} C_VEL
LIN {X 0,Y 429.368,Z 652.815,A -85,B 0,C 180,E1 -17472.364,E2 -17472.364} C_VEL
LIN {X 0,Y 429.999,Z 641.514,A -85,B 0,C 180,E1 -17473.542,E2 -17473.542} C_VEL
LIN {X 0,Y 430.768,Z 629.238,A -85,B 0,C 180,E1 -17474.598,E2 -17474.598} C_VEL
LIN {X 0,Y 431.601,Z 615.827,A -85,B 0,C 180,E1 -17475.532,E2 -17475.532} C_VEL
LIN {X 0,Y 432.069,Z 603.081,A -85,B 0,C 180,E1 -17476.239,E2 -17476.239} C_VEL
LIN {X 0,Y 432.662,Z 588.56,A -85,B 0,C 180,E1 -17476.852,E2 -17476.852} C_VEL
LIN {X 0,Y 433.207,Z 573.496,A -85,B 0,C 180,E1 -17477.287,E2 -17477.287} C_VEL
LIN {X 0,Y 435.82,Z 470.888,A -85,B 0,C 180,E1 -17479.603,E2 -17479.603} C_VEL
LIN {X 0,Y 432.847,Z 439.629,A -85,B 0,C 180,E1 -17480.424,E2 -17480.424} C_VEL
LIN {X 0,Y 434.465,Z 412.896,A -85,B 0,C 180,E1 -17483.769,E2 -17483.769} C_VEL
LIN {X 0,Y 436.232,Z 385.281,A -85,B 0,C 180,E1 -17487.234,E2 -17487.234} C_VEL
LIN {X 0,Y 436.732,Z 377.289,A -85,B 0,C 180,E1 -17488.24,E2 -17488.24} C_VEL
LIN {X 0,Y 432.871,Z 359.596,A -85,B 0,C 180,E1 -17490.685,E2 -17490.685} C_VEL
LIN {X 0,Y 429.469,Z 344.547,A -85,B 0,C 180,E1 -17492.84,E2 -17492.84} C_VEL
LIN {X 0,Y 429.424,Z 344.549,A -85,B 0,C 180,E1 -17495.959,E2 -17495.959} C_VEL
LIN {X 0,Y 429.439,Z 344.548,A -85,B 0,C 180,E1 -17499.503,E2 -17499.503} C_VEL
LIN {X 0,Y 429.436,Z 344.55,A -85,B 0,C 180,E1 -17502.778,E2 -17502.778} C_VEL
LIN {X 0,Y 429.42,Z 344.547,A -85,B 0,C 180,E1 -17505.866,E2 -17505.866} C_VEL
LIN {X 0,Y 429.442,Z 344.547,A -85,B 0,C 180,E1 -17509.275,E2 -17509.275} C_VEL
LIN {X 0,Y 429.416,Z 344.549,A -85,B 0,C 180,E1 -17511.696,E2 -17511.696} C_VEL
LIN {X 0,Y 429.431,Z 344.548,A -85,B 0,C 180,E1 -17515.188,E2 -17515.188} C_VEL
LIN {X 0,Y 429.418,Z 344.552,A -85,B 0,C 180,E1 -17518.536,E2 -17518.536} C_VEL
LIN {X 0,Y 429.449,Z 344.546,A -85,B 0,C 180,E1 -17521.771,E2 -17521.771} C_VEL
LIN {X 0,Y 429.412,Z 344.551,A -85,B 0,C 180,E1 -17524.906,E2 -17524.906} C_VEL
LIN {X 0,Y 429.473,Z 344.548,A -85,B 0,C 180,E1 -17528.379,E2 -17528.379} C_VEL
LIN {X 0,Y 429.496,Z 344.541,A -85,B 0,C 180,E1 -17531.067,E2 -17531.067} C_VEL
LIN {X 0,Y 429.486,Z 344.545,A -85,B 0,C 180,E1 -17533.641,E2 -17533.641} C_VEL
LIN {X 0,Y 431.871,Z 350.938,A -85,B 0,C 180,E1 -17533.886,E2 -17533.886} C_VEL
LIN {X 0,Y 438.875,Z 369.044,A -85,B 0,C 180,E1 -17534.525,E2 -17534.525} C_VEL
LIN {X 0,Y 437.695,Z 456.989,A -85,B 0,C 180,E1 -17535.963,E2 -17535.963} C_VEL
LIN {X 0,Y 437.587,Z 471.015,A -85,B 0,C 180,E1 -17536.284,E2 -17536.284} C_VEL
LIN {X 0,Y 437.243,Z 485.302,A -85,B 0,C 180,E1 -17536.804,E2 -17536.804} C_VEL
LIN {X 0,Y 436.571,Z 498.968,A -85,B 0,C 180,E1 -17537.491,E2 -17537.491} C_VEL
LIN {X 0,Y 435.844,Z 511.254,A -85,B 0,C 180,E1 -17538.294,E2 -17538.294} C_VEL
LIN {X 0,Y 435.114,Z 523.386,A -85,B 0,C 180,E1 -17539.291,E2 -17539.291} C_VEL
LIN {X 0,Y 434.071,Z 535.191,A -85,B 0,C 180,E1 -17540.48,E2 -17540.48} C_VEL
LIN {X 0,Y 433.107,Z 544.623,A -85,B 0,C 180,E1 -17541.631,E2 -17541.631} C_VEL
LIN {X 0,Y 432.066,Z 554.084,A -85,B 0,C 180,E1 -17543.016,E2 -17543.016} C_VEL
LIN {X 0,Y 431.197,Z 561.931,A -85,B 0,C 180,E1 -17544.407,E2 -17544.407} C_VEL
LIN {X 0,Y 430.449,Z 568.476,A -85,B 0,C 180,E1 -17545.801,E2 -17545.801} C_VEL
LIN {X 0,Y 429.872,Z 573.923,A -85,B 0,C 180,E1 -17547.198,E2 -17547.198} C_VEL
LIN {X 0,Y 429.339,Z 579.635,A -85,B 0,C 180,E1 -17549.065,E2 -17549.065} C_VEL
LIN {X 0,Y 428.969,Z 583.825,A -85,B 0,C 180,E1 -17550.936,E2 -17550.936} C_VEL
LIN {X 0,Y 428.85,Z 586.612,A -85,B 0,C 180,E1 -17552.809,E2 -17552.809} C_VEL
LIN {X 0,Y 428.839,Z 588.195,A -85,B 0,C 180,E1 -17554.896,E2 -17554.896} C_VEL
LIN {X 0,Y 428.95,Z 588.274,A -85,B 0,C 180,E1 -17556.564,E2 -17556.564} C_VEL
LIN {X 0,Y 429.206,Z 587.173,A -85,B 0,C 180,E1 -17558.446,E2 -17558.446} C_VEL
LIN {X 0,Y 429.624,Z 584.747,A -85,B 0,C 180,E1 -17560.332,E2 -17560.332} C_VEL
LIN {X 0,Y 430.46,Z 580.871,A -85,B 0,C 180,E1 -17562.213,E2 -17562.213} C_VEL
LIN {X 0,Y 431.36,Z 575.462,A -85,B 0,C 180,E1 -17564.098,E2 -17564.098} C_VEL
LIN {X 0,Y 432.265,Z 570.309,A -85,B 0,C 180,E1 -17565.508,E2 -17565.508} C_VEL
LIN {X 0,Y 433.266,Z 564.04,A -85,B 0,C 180,E1 -17566.918,E2 -17566.918} C_VEL
LIN {X 0,Y 434.459,Z 556.457,A -85,B 0,C 180,E1 -17568.324,E2 -17568.324} C_VEL
LIN {X 0,Y 435.769,Z 547.329,A -85,B 0,C 180,E1 -17569.728,E2 -17569.728} C_VEL
LIN {X 0,Y 436.555,Z 541.317,A -85,B 0,C 180,E1 -17570.517,E2 -17570.517} C_VEL
LIN {X 0,Y 436.465,Z 537.117,A -85,B 0,C 180,E1 -17571.057,E2 -17571.057} C_VEL
LIN {X 0,Y 434.572,Z 530.195,A -85,B 0,C 180,E1 -17571.953,E2 -17571.953} C_VEL
LIN {X 0,Y 432.719,Z 522.904,A -85,B 0,C 180,E1 -17572.803,E2 -17572.803} C_VEL
LIN {X 0,Y 432.651,Z 518.011,A -85,B 0,C 180,E1 -17573.252,E2 -17573.252} C_VEL
LIN {X 0,Y 433.824,Z 505.171,A -85,B 0,C 180,E1 -17574.186,E2 -17574.186} C_VEL
LIN {X 0,Y 434.371,Z 494.97,A -85,B 0,C 180,E1 -17574.788,E2 -17574.788} C_VEL
LIN {X 0,Y 435.047,Z 481.109,A -85,B 0,C 180,E1 -17575.417,E2 -17575.417} C_VEL
LIN {X 0,Y 435.396,Z 466.678,A -85,B 0,C 180,E1 -17575.873,E2 -17575.873} C_VEL
LIN {X 0,Y 436.094,Z 425.19,A -85,B 0,C 180,E1 -17576.598,E2 -17576.598} C_VEL
LIN {X 0,Y 437.073,Z 377.652,A -85,B 0,C 180,E1 -17577.383,E2 -17577.383} C_VEL
LIN {X 0,Y 426.511,Z 354.496,A -85,B 0,C 180,E1 -17578.477,E2 -17578.477} C_VEL
LIN {X 0,Y 422.589,Z 346.501,A -85,B 0,C 180,E1 -17578.888,E2 -17578.888} C_VEL
LIN {X 0,Y 422.39,Z 345.43,A -85,B 0,C 180,E1 -17578.941,E2 -17578.941} C_VEL
LIN {X 0,Y 422.316,Z 345.439,A -85,B 0,C 180,E1 -17582.233,E2 -17582.233} C_VEL
LIN {X 0,Y 422.296,Z 345.44,A -85,B 0,C 180,E1 -17585.635,E2 -17585.635} C_VEL
LIN {X 0,Y 422.32,Z 345.438,A -85,B 0,C 180,E1 -17588.782,E2 -17588.782} C_VEL
LIN {X 0,Y 422.317,Z 345.439,A -85,B 0,C 180,E1 -17591.724,E2 -17591.724} C_VEL
LIN {X 0,Y 422.359,Z 345.429,A -85,B 0,C 180,E1 -17594.51,E2 -17594.51} C_VEL
LIN {X 0,Y 422.337,Z 345.433,A -85,B 0,C 180,E1 -17597.157,E2 -17597.157} C_VEL
LIN {X 0,Y 422.353,Z 345.433,A -85,B 0,C 180,E1 -17599.719,E2 -17599.719} C_VEL
LIN {X 0,Y 422.323,Z 345.399,A -85,B 0,C 180,E1 -17603.339,E2 -17603.339} C_VEL
LIN {X 0,Y 422.316,Z 345.432,A -85,B 0,C 180,E1 -17606.815,E2 -17606.815} C_VEL
LIN {X 0,Y 422.353,Z 345.426,A -85,B 0,C 180,E1 -17610.163,E2 -17610.163} C_VEL
LIN {X 0,Y 422.405,Z 345.418,A -85,B 0,C 180,E1 -17613.566,E2 -17613.566} C_VEL
LIN {X 0,Y 422.339,Z 345.432,A -85,B 0,C 180,E1 -17616.544,E2 -17616.544} C_VEL
LIN {X 0,Y 422.412,Z 345.417,A -85,B 0,C 180,E1 -17619.219,E2 -17619.219} C_VEL
LIN {X 0,Y 428.371,Z 366.374,A -85,B 0,C 180,E1 -17619.883,E2 -17619.883} C_VEL
LIN {X 0,Y 426.221,Z 463.406,A -85,B 0,C 180,E1 -17622.11,E2 -17622.11} C_VEL
LIN {X 0,Y 426.028,Z 479.176,A -85,B 0,C 180,E1 -17622.678,E2 -17622.678} C_VEL
LIN {X 0,Y 425.517,Z 493.425,A -85,B 0,C 180,E1 -17623.38,E2 -17623.38} C_VEL
LIN {X 0,Y 425.031,Z 506.605,A -85,B 0,C 180,E1 -17624.221,E2 -17624.221} C_VEL
LIN {X 0,Y 424.327,Z 520.167,A -85,B 0,C 180,E1 -17625.297,E2 -17625.297} C_VEL
LIN {X 0,Y 423.734,Z 532.493,A -85,B 0,C 180,E1 -17626.497,E2 -17626.497} C_VEL
LIN {X 0,Y 423.291,Z 543.625,A -85,B 0,C 180,E1 -17627.82,E2 -17627.82} C_VEL
LIN {X 0,Y 422.71,Z 553.693,A -85,B 0,C 180,E1 -17629.256,E2 -17629.256} C_VEL
LIN {X 0,Y 422.217,Z 562.07,A -85,B 0,C 180,E1 -17630.691,E2 -17630.691} C_VEL
LIN {X 0,Y 421.882,Z 570.122,A -85,B 0,C 180,E1 -17632.367,E2 -17632.367} C_VEL
LIN {X 0,Y 421.667,Z 575.713,A -85,B 0,C 180,E1 -17633.801,E2 -17633.801} C_VEL
LIN {X 0,Y 421.587,Z 580.953,A -85,B 0,C 180,E1 -17635.469,E2 -17635.469} C_VEL
LIN {X 0,Y 421.607,Z 584.934,A -85,B 0,C 180,E1 -17637.143,E2 -17637.143} C_VEL
LIN {X 0,Y 421.755,Z 588.006,A -85,B 0,C 180,E1 -17639.048,E2 -17639.048} C_VEL
LIN {X 0,Y 422.019,Z 589.626,A -85,B 0,C 180,E1 -17640.951,E2 -17640.951} C_VEL
LIN {X 0,Y 422.532,Z 589.817,A -85,B 0,C 180,E1 -17642.85,E2 -17642.85} C_VEL
LIN {X 0,Y 423.341,Z 588.569,A -85,B 0,C 180,E1 -17644.745,E2 -17644.745} C_VEL
LIN {X 0,Y 424.289,Z 585.845,A -85,B 0,C 180,E1 -17646.636,E2 -17646.636} C_VEL
LIN {X 0,Y 425.213,Z 582.797,A -85,B 0,C 180,E1 -17648.049,E2 -17648.049} C_VEL
LIN {X 0,Y 426.454,Z 578.774,A -85,B 0,C 180,E1 -17649.453,E2 -17649.453} C_VEL
LIN {X 0,Y 427.706,Z 573.79,A -85,B 0,C 180,E1 -17650.855,E2 -17650.855} C_VEL
LIN {X 0,Y 429.276,Z 566.611,A -85,B 0,C 180,E1 -17652.486,E2 -17652.486} C_VEL
LIN {X 0,Y 430.846,Z 559.047,A -85,B 0,C 180,E1 -17653.874,E2 -17653.874} C_VEL
LIN {X 0,Y 432.486,Z 549.964,A -85,B 0,C 180,E1 -17655.259,E2 -17655.259} C_VEL
LIN {X 0,Y 434.182,Z 539.903,A -85,B 0,C 180,E1 -17656.519,E2 -17656.519} C_VEL
LIN {X 0,Y 435.897,Z 528.836,A -85,B 0,C 180,E1 -17657.656,E2 -17657.656} C_VEL
LIN {X 0,Y 437.491,Z 516.847,A -85,B 0,C 180,E1 -17658.675,E2 -17658.675} C_VEL
LIN {X 0,Y 438.873,Z 503.75,A -85,B 0,C 180,E1 -17659.582,E2 -17659.582} C_VEL
LIN {X 0,Y 440.003,Z 489.206,A -85,B 0,C 180,E1 -17660.367,E2 -17660.367} C_VEL
LIN {X 0,Y 440.852,Z 474.861,A -85,B 0,C 180,E1 -17660.946,E2 -17660.946} C_VEL
LIN {X 0,Y 441.795,Z 454.183,A -85,B 0,C 180,E1 -17661.539,E2 -17661.539} C_VEL
LIN {X 0,Y 446.618,Z 385.822,A -85,B 0,C 180,E1 -17663.361,E2 -17663.361} C_VEL
LIN {X 0,Y 441.434,Z 375.716,A -85,B 0,C 180,E1 -17664.382,E2 -17664.382} C_VEL
LIN {X 0,Y 435.925,Z 366.449,A -85,B 0,C 180,E1 -17665.509,E2 -17665.509} C_VEL
LIN {X 0,Y 431.038,Z 358.746,A -85,B 0,C 180,E1 -17666.598,E2 -17666.598} C_VEL
LIN {X 0,Y 428.482,Z 354.954,A -85,B 0,C 180,E1 -17667.19,E2 -17667.19} C_VEL
LIN {X 0,Y 426.307,Z 351.952,A -85,B 0,C 180,E1 -17667.711,E2 -17667.711} C_VEL
LIN {X 0,Y 425.575,Z 350.469,A -85,B 0,C 180,E1 -17667.923,E2 -17667.923} C_VEL
LIN {X 0,Y 423.452,Z 348.335,A -85,B 0,C 180,E1 -17668.435,E2 -17668.435} C_VEL
LIN {X 0,Y 422.459,Z 345.875,A -85,B 0,C 180,E1 -17668.756,E2 -17668.756} C_VEL
LIN {X 0,Y 422.379,Z 345.429,A -85,B 0,C 180,E1 -17668.813,E2 -17668.813} C_VEL
LIN {X 0,Y 422.368,Z 345.428,A -85,B 0,C 180,E1 -17672.245,E2 -17672.245} C_VEL
LIN {X 0,Y 422.398,Z 345.42,A -85,B 0,C 180,E1 -17675.654,E2 -17675.654} C_VEL
LIN {X 0,Y 422.338,Z 345.425,A -85,B 0,C 180,E1 -17679.067,E2 -17679.067} C_VEL
LIN {X 0,Y 422.328,Z 345.429,A -85,B 0,C 180,E1 -17681.725,E2 -17681.725} C_VEL
LIN {X 0,Y 422.361,Z 345.426,A -85,B 0,C 180,E1 -17684.511,E2 -17684.511} C_VEL
LIN {X 0,Y 422.335,Z 345.436,A -85,B 0,C 180,E1 -17687.157,E2 -17687.157} C_VEL
LIN {X 0,Y 422.35,Z 345.43,A -85,B 0,C 180,E1 -17689.719,E2 -17689.719} C_VEL
LIN {X 0,Y 422.316,Z 345.436,A -85,B 0,C 180,E1 -17693.338,E2 -17693.338} C_VEL
LIN {X 0,Y 422.326,Z 345.564,A -85,B 0,C 180,E1 -17694.951,E2 -17694.951} C_VEL
LIN {X 0,Y 426.16,Z 360.221,A -85,B 0,C 180,E1 -17697.712,E2 -17697.712} C_VEL
LIN {X 0,Y 429.729,Z 376.024,A -85,B 0,C 180,E1 -17700.519,E2 -17700.519} C_VEL
LIN {X 0,Y 430.337,Z 380.981,A -85,B 0,C 180,E1 -17701.346,E2 -17701.346} C_VEL
LIN {X 0,Y 430.379,Z 382.431,A -85,B 0,C 180,E1 -17701.473,E2 -17701.473} C_VEL
LIN {X 0,Y 431.739,Z 391.288,A -85,B 0,C 180,E1 -17702.065,E2 -17702.065} C_VEL
LIN {X 0,Y 433.889,Z 404.467,A -85,B 0,C 180,E1 -17702.903,E2 -17702.903} C_VEL
LIN {X 0,Y 436.764,Z 424.819,A -85,B 0,C 180,E1 -17704.073,E2 -17704.073} C_VEL
LIN {X 0,Y 438.602,Z 440.486,A -85,B 0,C 180,E1 -17704.874,E2 -17704.874} C_VEL
LIN {X 0,Y 440.052,Z 456.103,A -85,B 0,C 180,E1 -17705.582,E2 -17705.582} C_VEL
LIN {X 0,Y 440.87,Z 477.894,A -85,B 0,C 180,E1 -17706.423,E2 -17706.423} C_VEL
LIN {X 0,Y 436.122,Z 551.037,A -85,B 0,C 180,E1 -17708.352,E2 -17708.352} C_VEL
LIN {X 0,Y 434.678,Z 566.273,A -85,B 0,C 180,E1 -17708.927,E2 -17708.927} C_VEL
LIN {X 0,Y 432.809,Z 580.763,A -85,B 0,C 180,E1 -17709.638,E2 -17709.638} C_VEL
LIN {X 0,Y 430.731,Z 594.68,A -85,B 0,C 180,E1 -17710.527,E2 -17710.527} C_VEL
LIN {X 0,Y 428.658,Z 608.209,A -85,B 0,C 180,E1 -17711.62,E2 -17711.62} C_VEL
LIN {X 0,Y 426.712,Z 620.263,A -85,B 0,C 180,E1 -17712.814,E2 -17712.814} C_VEL
LIN {X 0,Y 424.861,Z 631.841,A -85,B 0,C 180,E1 -17714.215,E2 -17714.215} C_VEL
LIN {X 0,Y 423.429,Z 641.956,A -85,B 0,C 180,E1 -17715.633,E2 -17715.633} C_VEL
LIN {X 0,Y 422.444,Z 650.53,A -85,B 0,C 180,E1 -17717.065,E2 -17717.065} C_VEL
LIN {X 0,Y 422.119,Z 653.934,A -85,B 0,C 180,E1 -17717.664,E2 -17717.664} C_VEL
LIN {X 0,Y 421.46,Z 663.424,A -85,B 0,C 180,E1 -17718.842,E2 -17718.842} C_VEL
LIN {X 0,Y 421.148,Z 670.974,A -85,B 0,C 180,E1 -17719.942,E2 -17719.942} C_VEL
LIN {X 0,Y 420.777,Z 679.371,A -85,B 0,C 180,E1 -17721.383,E2 -17721.383} C_VEL
LIN {X 0,Y 420.495,Z 687.377,A -85,B 0,C 180,E1 -17723.063,E2 -17723.063} C_VEL
LIN {X 0,Y 420.364,Z 693.715,A -85,B 0,C 180,E1 -17724.742,E2 -17724.742} C_VEL
LIN {X 0,Y 420.283,Z 697.965,A -85,B 0,C 180,E1 -17726.177,E2 -17726.177} C_VEL
LIN {X 0,Y 420.239,Z 700.279,A -85,B 0,C 180,E1 -17727.134,E2 -17727.134} C_VEL
LIN {X 0,Y 420.259,Z 702.164,A -85,B 0,C 180,E1 -17728.09,E2 -17728.09} C_VEL
LIN {X 0,Y 420.228,Z 704.735,A -85,B 0,C 180,E1 -17730,E2 -17730} C_VEL
LIN {X 0,Y 420.245,Z 705.818,A -85,B 0,C 180,E1 -17731.91,E2 -17731.91} C_VEL
LIN {X 0,Y 420.307,Z 705.432,A -85,B 0,C 180,E1 -17733.822,E2 -17733.822} C_VEL
LIN {X 0,Y 420.59,Z 703.593,A -85,B 0,C 180,E1 -17735.735,E2 -17735.735} C_VEL
LIN {X 0,Y 421.098,Z 700.27,A -85,B 0,C 180,E1 -17737.647,E2 -17737.647} C_VEL
LIN {X 0,Y 421.694,Z 696.723,A -85,B 0,C 180,E1 -17739.079,E2 -17739.079} C_VEL
LIN {X 0,Y 422.459,Z 692.26,A -85,B 0,C 180,E1 -17740.508,E2 -17740.508} C_VEL
LIN {X 0,Y 423.784,Z 685.747,A -85,B 0,C 180,E1 -17742.165,E2 -17742.165} C_VEL
LIN {X 0,Y 425.164,Z 677.709,A -85,B 0,C 180,E1 -17743.821,E2 -17743.821} C_VEL
LIN {X 0,Y 427.062,Z 667.776,A -85,B 0,C 180,E1 -17745.457,E2 -17745.457} C_VEL
LIN {X 0,Y 428.879,Z 657.409,A -85,B 0,C 180,E1 -17746.851,E2 -17746.851} C_VEL
LIN {X 0,Y 431.011,Z 644.827,A -85,B 0,C 180,E1 -17748.23,E2 -17748.23} C_VEL
LIN {X 0,Y 433.033,Z 631.99,A -85,B 0,C 180,E1 -17749.365,E2 -17749.365} C_VEL
LIN {X 0,Y 435.009,Z 617.608,A -85,B 0,C 180,E1 -17750.377,E2 -17750.377} C_VEL
LIN {X 0,Y 436.745,Z 603.503,A -85,B 0,C 180,E1 -17751.152,E2 -17751.152} C_VEL
LIN {X 0,Y 438.353,Z 587.95,A -85,B 0,C 180,E1 -17751.777,E2 -17751.777} C_VEL
LIN {X 0,Y 440.552,Z 558.048,A -85,B 0,C 180,E1 -17752.601,E2 -17752.601} C_VEL
LIN {X 0,Y 446.37,Z 480.154,A -85,B 0,C 180,E1 -17754.734,E2 -17754.734} C_VEL
LIN {X 0,Y 446.111,Z 465.963,A -85,B 0,C 180,E1 -17755.301,E2 -17755.301} C_VEL
LIN {X 0,Y 444.764,Z 446.512,A -85,B 0,C 180,E1 -17756.237,E2 -17756.237} C_VEL
LIN {X 0,Y 443.774,Z 437.294,A -85,B 0,C 180,E1 -17756.744,E2 -17756.744} C_VEL
LIN {X 0,Y 444.294,Z 417.882,A -85,B 0,C 180,E1 -17758.388,E2 -17758.388} C_VEL
LIN {X 0,Y 444.773,Z 403.923,A -85,B 0,C 180,E1 -17759.753,E2 -17759.753} C_VEL
LIN {X 0,Y 445.409,Z 394.3,A -85,B 0,C 180,E1 -17760.764,E2 -17760.764} C_VEL
LIN {X 0,Y 445.25,Z 389.644,A -85,B 0,C 180,E1 -17761.402,E2 -17761.402} C_VEL
LIN {X 0,Y 444.616,Z 382.36,A -85,B 0,C 180,E1 -17762.618,E2 -17762.618} C_VEL
LIN {X 0,Y 443.008,Z 379.238,A -85,B 0,C 180,E1 -17763.6,E2 -17763.6} C_VEL
LIN {X 0,Y 441.102,Z 375.958,A -85,B 0,C 180,E1 -17764.866,E2 -17764.866} C_VEL
LIN {X 0,Y 438.537,Z 371.828,A -85,B 0,C 180,E1 -17767.002,E2 -17767.002} C_VEL
LIN {X 0,Y 437.096,Z 369.833,A -85,B 0,C 180,E1 -17768.68,E2 -17768.68} C_VEL
LIN {X 0,Y 435.89,Z 368.512,A -85,B 0,C 180,E1 -17770.952,E2 -17770.952} C_VEL
LIN {X 0,Y 435.632,Z 368.368,A -85,B 0,C 180,E1 -17772.478,E2 -17772.478} C_VEL
LIN {X 0,Y 436.129,Z 369.36,A -85,B 0,C 180,E1 -17774.964,E2 -17774.964} C_VEL
LIN {X 0,Y 436.636,Z 370.901,A -85,B 0,C 180,E1 -17776.386,E2 -17776.386} C_VEL
LIN {X 0,Y 438.074,Z 374.529,A -85,B 0,C 180,E1 -17778.72,E2 -17778.72} C_VEL
LIN {X 0,Y 439.724,Z 379.211,A -85,B 0,C 180,E1 -17780.822,E2 -17780.822} C_VEL
LIN {X 0,Y 441.785,Z 385.198,A -85,B 0,C 180,E1 -17782.952,E2 -17782.952} C_VEL
LIN {X 0,Y 443.72,Z 392.254,A -85,B 0,C 180,E1 -17784.959,E2 -17784.959} C_VEL
LIN {X 0,Y 445.409,Z 400.257,A -85,B 0,C 180,E1 -17786.866,E2 -17786.866} C_VEL
LIN {X 0,Y 446.432,Z 407.087,A -85,B 0,C 180,E1 -17788.283,E2 -17788.283} C_VEL
LIN {X 0,Y 444.404,Z 418.722,A -85,B 0,C 180,E1 -17789.958,E2 -17789.958} C_VEL
LIN {X 0,Y 440.905,Z 439.858,A -85,B 0,C 180,E1 -17792.878,E2 -17792.878} C_VEL
LIN {X 0,Y 444.142,Z 457.98,A -85,B 0,C 180,E1 -17794.054,E2 -17794.054} C_VEL
LIN {X 0,Y 446.442,Z 475.227,A -85,B 0,C 180,E1 -17794.999,E2 -17794.999} C_VEL
LIN {X 0,Y 446.762,Z 480.163,A -85,B 0,C 180,E1 -17795.219,E2 -17795.219} C_VEL
LIN {X 0,Y 440.58,Z 563.645,A -85,B 0,C 180,E1 -17797.459,E2 -17797.459} C_VEL
LIN {X 0,Y 438.922,Z 585.439,A -85,B 0,C 180,E1 -17798.074,E2 -17798.074} C_VEL
LIN {X 0,Y 437.334,Z 600.698,A -85,B 0,C 180,E1 -17798.693,E2 -17798.693} C_VEL
LIN {X 0,Y 435.727,Z 613.974,A -85,B 0,C 180,E1 -17799.412,E2 -17799.412} C_VEL
LIN {X 0,Y 433.695,Z 628.488,A -85,B 0,C 180,E1 -17800.42,E2 -17800.42} C_VEL
LIN {X 0,Y 431.662,Z 641.537,A -85,B 0,C 180,E1 -17801.554,E2 -17801.554} C_VEL
LIN {X 0,Y 429.853,Z 652.349,A -85,B 0,C 180,E1 -17802.7,E2 -17802.7} C_VEL
LIN {X 0,Y 427.848,Z 663.216,A -85,B 0,C 180,E1 -17804.085,E2 -17804.085} C_VEL
LIN {X 0,Y 425.904,Z 673.582,A -85,B 0,C 180,E1 -17805.718,E2 -17805.718} C_VEL
LIN {X 0,Y 424.373,Z 682.054,A -85,B 0,C 180,E1 -17807.368,E2 -17807.368} C_VEL
LIN {X 0,Y 423.006,Z 688.919,A -85,B 0,C 180,E1 -17809.023,E2 -17809.023} C_VEL
LIN {X 0,Y 422.07,Z 693.645,A -85,B 0,C 180,E1 -17810.448,E2 -17810.448} C_VEL
LIN {X 0,Y 421.171,Z 698.526,A -85,B 0,C 180,E1 -17812.355,E2 -17812.355} C_VEL
LIN {X 0,Y 420.585,Z 701.83,A -85,B 0,C 180,E1 -17814.265,E2 -17814.265} C_VEL
LIN {X 0,Y 420.277,Z 703.653,A -85,B 0,C 180,E1 -17816.178,E2 -17816.178} C_VEL
LIN {X 0,Y 420.179,Z 704.04,A -85,B 0,C 180,E1 -17818.09,E2 -17818.09} C_VEL
LIN {X 0,Y 420.153,Z 702.975,A -85,B 0,C 180,E1 -17820,E2 -17820} C_VEL
LIN {X 0,Y 420.179,Z 700.442,A -85,B 0,C 180,E1 -17821.911,E2 -17821.911} C_VEL
LIN {X 0,Y 420.17,Z 697.485,A -85,B 0,C 180,E1 -17823.345,E2 -17823.345} C_VEL
LIN {X 0,Y 420.296,Z 693.627,A -85,B 0,C 180,E1 -17824.78,E2 -17824.78} C_VEL
LIN {X 0,Y 420.401,Z 688.766,A -85,B 0,C 180,E1 -17826.218,E2 -17826.218} C_VEL
LIN {X 0,Y 420.667,Z 681.646,A -85,B 0,C 180,E1 -17827.896,E2 -17827.896} C_VEL
LIN {X 0,Y 421.17,Z 672.798,A -85,B 0,C 180,E1 -17829.574,E2 -17829.574} C_VEL
LIN {X 0,Y 421.636,Z 663.649,A -85,B 0,C 180,E1 -17830.996,E2 -17830.996} C_VEL
LIN {X 0,Y 422.26,Z 653.33,A -85,B 0,C 180,E1 -17832.332,E2 -17832.332} C_VEL
LIN {X 0,Y 422.923,Z 642.155,A -85,B 0,C 180,E1 -17833.529,E2 -17833.529} C_VEL
LIN {X 0,Y 423.651,Z 629.982,A -85,B 0,C 180,E1 -17834.604,E2 -17834.604} C_VEL
LIN {X 0,Y 424.487,Z 616.731,A -85,B 0,C 180,E1 -17835.554,E2 -17835.554} C_VEL
LIN {X 0,Y 425.015,Z 604.246,A -85,B 0,C 180,E1 -17836.271,E2 -17836.271} C_VEL
LIN {X 0,Y 425.588,Z 589.401,A -85,B 0,C 180,E1 -17836.924,E2 -17836.924} C_VEL
LIN {X 0,Y 426.111,Z 575.207,A -85,B 0,C 180,E1 -17837.357,E2 -17837.357} C_VEL
LIN {X 0,Y 428.762,Z 470.838,A -85,B 0,C 180,E1 -17839.784,E2 -17839.784} C_VEL
LIN {X 0,Y 425.869,Z 439.563,A -85,B 0,C 180,E1 -17840.627,E2 -17840.627} C_VEL
LIN {X 0,Y 427.629,Z 411.533,A -85,B 0,C 180,E1 -17844.173,E2 -17844.173} C_VEL
LIN {X 0,Y 429.487,Z 383.746,A -85,B 0,C 180,E1 -17847.698,E2 -17847.698} C_VEL
LIN {X 0,Y 429.811,Z 378.589,A -85,B 0,C 180,E1 -17848.356,E2 -17848.356} C_VEL
LIN {X 0,Y 425.481,Z 358.839,A -85,B 0,C 180,E1 -17851.125,E2 -17851.125} C_VEL
LIN {X 0,Y 422.404,Z 345.428,A -85,B 0,C 180,E1 -17853.074,E2 -17853.074} C_VEL
LIN {X 0,Y 422.407,Z 345.426,A -85,B 0,C 180,E1 -17855.656,E2 -17855.656} C_VEL
LIN {X 0,Y 422.374,Z 345.433,A -85,B 0,C 180,E1 -17859.063,E2 -17859.063} C_VEL
LIN {X 0,Y 422.364,Z 345.428,A -85,B 0,C 180,E1 -17861.731,E2 -17861.731} C_VEL
LIN {X 0,Y 422.38,Z 345.427,A -85,B 0,C 180,E1 -17864.514,E2 -17864.514} C_VEL
LIN {X 0,Y 422.39,Z 345.428,A -85,B 0,C 180,E1 -17867.164,E2 -17867.164} C_VEL
LIN {X 0,Y 422.388,Z 345.423,A -85,B 0,C 180,E1 -17869.714,E2 -17869.714} C_VEL
LIN {X 0,Y 422.359,Z 345.434,A -85,B 0,C 180,E1 -17872.754,E2 -17872.754} C_VEL
LIN {X 0,Y 422.389,Z 345.425,A -85,B 0,C 180,E1 -17876.012,E2 -17876.012} C_VEL
LIN {X 0,Y 422.375,Z 345.426,A -85,B 0,C 180,E1 -17879.064,E2 -17879.064} C_VEL
LIN {X 0,Y 422.403,Z 345.428,A -85,B 0,C 180,E1 -17882.335,E2 -17882.335} C_VEL
LIN {X 0,Y 422.381,Z 345.427,A -85,B 0,C 180,E1 -17885.795,E2 -17885.795} C_VEL
LIN {X 0,Y 422.427,Z 345.424,A -85,B 0,C 180,E1 -17888.605,E2 -17888.605} C_VEL
LIN {X 0,Y 422.437,Z 345.422,A -85,B 0,C 180,E1 -17891.637,E2 -17891.637} C_VEL
LIN {X 0,Y 422.425,Z 345.424,A -85,B 0,C 180,E1 -17893.318,E2 -17893.318} C_VEL
LIN {X 0,Y 424.935,Z 352.037,A -85,B 0,C 180,E1 -17893.567,E2 -17893.567} C_VEL
LIN {X 0,Y 432.097,Z 370.561,A -85,B 0,C 180,E1 -17894.236,E2 -17894.236} C_VEL
LIN {X 0,Y 430.925,Z 460.381,A -85,B 0,C 180,E1 -17895.738,E2 -17895.738} C_VEL
LIN {X 0,Y 430.757,Z 475.116,A -85,B 0,C 180,E1 -17896.123,E2 -17896.123} C_VEL
LIN {X 0,Y 430.329,Z 488.445,A -85,B 0,C 180,E1 -17896.648,E2 -17896.648} C_VEL
LIN {X 0,Y 429.749,Z 500.559,A -85,B 0,C 180,E1 -17897.289,E2 -17897.289} C_VEL
LIN {X 0,Y 429.014,Z 512.671,A -85,B 0,C 180,E1 -17898.105,E2 -17898.105} C_VEL
LIN {X 0,Y 428.233,Z 524.687,A -85,B 0,C 180,E1 -17899.117,E2 -17899.117} C_VEL
LIN {X 0,Y 427.151,Z 536.4,A -85,B 0,C 180,E1 -17900.324,E2 -17900.324} C_VEL
LIN {X 0,Y 426.175,Z 545.757,A -85,B 0,C 180,E1 -17901.494,E2 -17901.494} C_VEL
LIN {X 0,Y 425.104,Z 555.157,A -85,B 0,C 180,E1 -17902.902,E2 -17902.902} C_VEL
LIN {X 0,Y 424.203,Z 562.952,A -85,B 0,C 180,E1 -17904.314,E2 -17904.314} C_VEL
LIN {X 0,Y 423.433,Z 569.451,A -85,B 0,C 180,E1 -17905.731,E2 -17905.731} C_VEL
LIN {X 0,Y 422.849,Z 574.856,A -85,B 0,C 180,E1 -17907.152,E2 -17907.152} C_VEL
LIN {X 0,Y 422.311,Z 580.528,A -85,B 0,C 180,E1 -17909.05,E2 -17909.05} C_VEL
LIN {X 0,Y 421.925,Z 584.684,A -85,B 0,C 180,E1 -17910.951,E2 -17910.951} C_VEL
LIN {X 0,Y 421.781,Z 587.44,A -85,B 0,C 180,E1 -17912.856,E2 -17912.856} C_VEL
LIN {X 0,Y 421.793,Z 588.936,A -85,B 0,C 180,E1 -17914.87,E2 -17914.87} C_VEL
LIN {X 0,Y 421.904,Z 589.036,A -85,B 0,C 180,E1 -17916.674,E2 -17916.674} C_VEL
LIN {X 0,Y 422.199,Z 587.899,A -85,B 0,C 180,E1 -17918.587,E2 -17918.587} C_VEL
LIN {X 0,Y 422.638,Z 585.43,A -85,B 0,C 180,E1 -17920.504,E2 -17920.504} C_VEL
LIN {X 0,Y 423.493,Z 581.513,A -85,B 0,C 180,E1 -17922.417,E2 -17922.417} C_VEL
LIN {X 0,Y 424.473,Z 576.062,A -85,B 0,C 180,E1 -17924.331,E2 -17924.331} C_VEL
LIN {X 0,Y 425.417,Z 570.867,A -85,B 0,C 180,E1 -17925.764,E2 -17925.764} C_VEL
LIN {X 0,Y 426.695,Z 563.192,A -85,B 0,C 180,E1 -17927.467,E2 -17927.467} C_VEL
LIN {X 0,Y 428.105,Z 554.037,A -85,B 0,C 180,E1 -17929.101,E2 -17929.101} C_VEL
LIN {X 0,Y 429.557,Z 544.223,A -85,B 0,C 180,E1 -17930.523,E2 -17930.523} C_VEL
LIN {X 0,Y 430.965,Z 533.271,A -85,B 0,C 180,E1 -17931.826,E2 -17931.826} C_VEL
LIN {X 0,Y 432.209,Z 522.338,A -85,B 0,C 180,E1 -17932.889,E2 -17932.889} C_VEL
LIN {X 0,Y 432.651,Z 518.011,A -85,B 0,C 180,E1 -17933.252,E2 -17933.252} C_VEL
LIN {X 0,Y 432.557,Z 513.058,A -85,B 0,C 180,E1 -17933.681,E2 -17933.681} C_VEL
LIN {X 0,Y 430.566,Z 505.007,A -85,B 0,C 180,E1 -17934.407,E2 -17934.407} C_VEL
LIN {X 0,Y 428.437,Z 496.653,A -85,B 0,C 180,E1 -17935.061,E2 -17935.061} C_VEL
LIN {X 0,Y 428.109,Z 491.23,A -85,B 0,C 180,E1 -17935.37,E2 -17935.37} C_VEL
LIN {X 0,Y 428.693,Z 477.299,A -85,B 0,C 180,E1 -17935.944,E2 -17935.944} C_VEL
LIN {X 0,Y 428.959,Z 463.96,A -85,B 0,C 180,E1 -17936.318,E2 -17936.318} C_VEL
LIN {X 0,Y 430.566,Z 379.427,A -85,B 0,C 180,E1 -17937.758,E2 -17937.758} C_VEL
LIN {X 0,Y 420.848,Z 358.122,A -85,B 0,C 180,E1 -17938.79,E2 -17938.79} C_VEL
LIN {X 0,Y 415.484,Z 347.088,A -85,B 0,C 180,E1 -17939.37,E2 -17939.37} C_VEL
LIN {X 0,Y 415.36,Z 346.307,A -85,B 0,C 180,E1 -17939.417,E2 -17939.417} C_VEL
LIN {X 0,Y 415.273,Z 346.314,A -85,B 0,C 180,E1 -17942.667,E2 -17942.667} C_VEL
LIN {X 0,Y 415.252,Z 346.317,A -85,B 0,C 180,E1 -17946.184,E2 -17946.184} C_VEL
LIN {X 0,Y 415.274,Z 346.314,A -85,B 0,C 180,E1 -17949.114,E2 -17949.114} C_VEL
LIN {X 0,Y 415.272,Z 346.316,A -85,B 0,C 180,E1 -17952.43,E2 -17952.43} C_VEL
LIN {X 0,Y 415.304,Z 346.306,A -85,B 0,C 180,E1 -17955.102,E2 -17955.102} C_VEL
LIN {X 0,Y 415.281,Z 346.31,A -85,B 0,C 180,E1 -17957.914,E2 -17957.914} C_VEL
LIN {X 0,Y 415.286,Z 346.299,A -85,B 0,C 180,E1 -17961.386,E2 -17961.386} C_VEL
LIN {X 0,Y 415.255,Z 346.282,A -85,B 0,C 180,E1 -17964.063,E2 -17964.063} C_VEL
LIN {X 0,Y 415.287,Z 346.311,A -85,B 0,C 180,E1 -17967.494,E2 -17967.494} C_VEL
LIN {X 0,Y 415.348,Z 346.294,A -85,B 0,C 180,E1 -17969.607,E2 -17969.607} C_VEL
LIN {X 0,Y 415.327,Z 346.302,A -85,B 0,C 180,E1 -17972.912,E2 -17972.912} C_VEL
LIN {X 0,Y 415.322,Z 346.309,A -85,B 0,C 180,E1 -17976.123,E2 -17976.123} C_VEL
LIN {X 0,Y 415.366,Z 346.294,A -85,B 0,C 180,E1 -17979.055,E2 -17979.055} C_VEL
LIN {X 0,Y 421.381,Z 367.744,A -85,B 0,C 180,E1 -17979.74,E2 -17979.74} C_VEL
LIN {X 0,Y 419.202,Z 464.35,A -85,B 0,C 180,E1 -17982.015,E2 -17982.015} C_VEL
LIN {X 0,Y 418.937,Z 479.743,A -85,B 0,C 180,E1 -17982.579,E2 -17982.579} C_VEL
LIN {X 0,Y 418.482,Z 493.803,A -85,B 0,C 180,E1 -17983.281,E2 -17983.281} C_VEL
LIN {X 0,Y 417.915,Z 507.88,A -85,B 0,C 180,E1 -17984.195,E2 -17984.195} C_VEL
LIN {X 0,Y 417.256,Z 521.357,A -85,B 0,C 180,E1 -17985.291,E2 -17985.291} C_VEL
LIN {X 0,Y 416.673,Z 533.6,A -85,B 0,C 180,E1 -17986.512,E2 -17986.512} C_VEL
LIN {X 0,Y 416.173,Z 544.84,A -85,B 0,C 180,E1 -17987.878,E2 -17987.878} C_VEL
LIN {X 0,Y 415.602,Z 554.703,A -85,B 0,C 180,E1 -17989.316,E2 -17989.316} C_VEL
LIN {X 0,Y 415.135,Z 563.068,A -85,B 0,C 180,E1 -17990.776,E2 -17990.776} C_VEL
LIN {X 0,Y 414.781,Z 571.113,A -85,B 0,C 180,E1 -17992.48,E2 -17992.48} C_VEL
LIN {X 0,Y 414.544,Z 577.527,A -85,B 0,C 180,E1 -17994.181,E2 -17994.181} C_VEL
LIN {X 0,Y 414.547,Z 583.15,A -85,B 0,C 180,E1 -17996.124,E2 -17996.124} C_VEL
LIN {X 0,Y 414.555,Z 587.2,A -85,B 0,C 180,E1 -17998.063,E2 -17998.063} C_VEL
LIN {X 0,Y 414.697,Z 588.656,A -85,B 0,C 180,E1 -17999.032,E2 -17999.032} C_VEL
LIN {X 0,Y 414.974,Z 590.442,A -85,B 0,C 180,E1 -18000.967,E2 -18000.967} C_VEL
LIN {X 0,Y 415.529,Z 590.786,A -85,B 0,C 180,E1 -18002.898,E2 -18002.898} C_VEL
LIN {X 0,Y 416.359,Z 589.693,A -85,B 0,C 180,E1 -18004.825,E2 -18004.825} C_VEL
LIN {X 0,Y 417.364,Z 587.178,A -85,B 0,C 180,E1 -18006.746,E2 -18006.746} C_VEL
LIN {X 0,Y 418.34,Z 584.245,A -85,B 0,C 180,E1 -18008.182,E2 -18008.182} C_VEL
LIN {X 0,Y 420.091,Z 578.909,A -85,B 0,C 180,E1 -18010.083,E2 -18010.083} C_VEL
LIN {X 0,Y 421.395,Z 573.762,A -85,B 0,C 180,E1 -18011.505,E2 -18011.505} C_VEL
LIN {X 0,Y 423.124,Z 566.314,A -85,B 0,C 180,E1 -18013.157,E2 -18013.157} C_VEL
LIN {X 0,Y 424.824,Z 558.506,A -85,B 0,C 180,E1 -18014.563,E2 -18014.563} C_VEL
LIN {X 0,Y 426.574,Z 549.106,A -85,B 0,C 180,E1 -18015.964,E2 -18015.964} C_VEL
LIN {X 0,Y 428.644,Z 537.675,A -85,B 0,C 180,E1 -18017.351,E2 -18017.351} C_VEL
LIN {X 0,Y 430.477,Z 525.99,A -85,B 0,C 180,E1 -18018.499,E2 -18018.499} C_VEL
LIN {X 0,Y 432.332,Z 511.839,A -85,B 0,C 180,E1 -18019.622,E2 -18019.622} C_VEL
LIN {X 0,Y 433.549,Z 499.135,A -85,B 0,C 180,E1 -18020.437,E2 -18020.437} C_VEL
LIN {X 0,Y 434.727,Z 483.551,A -85,B 0,C 180,E1 -18021.193,E2 -18021.193} C_VEL
LIN {X 0,Y 435.49,Z 467.932,A -85,B 0,C 180,E1 -18021.742,E2 -18021.742} C_VEL
LIN {X 0,Y 439.321,Z 412.888,A -85,B 0,C 180,E1 -18023.24,E2 -18023.24} C_VEL
LIN {X 0,Y 441.281,Z 388.767,A -85,B 0,C 180,E1 -18023.899,E2 -18023.899} C_VEL
LIN {X 0,Y 436.075,Z 378.618,A -85,B 0,C 180,E1 -18024.988,E2 -18024.988} C_VEL
LIN {X 0,Y 430.241,Z 368.786,A -85,B 0,C 180,E1 -18026.267,E2 -18026.267} C_VEL
LIN {X 0,Y 424.989,Z 360.697,A -85,B 0,C 180,E1 -18027.511,E2 -18027.511} C_VEL
LIN {X 0,Y 422.634,Z 357.182,A -85,B 0,C 180,E1 -18028.127,E2 -18028.127} C_VEL
LIN {X 0,Y 421.466,Z 355.768,A -85,B 0,C 180,E1 -18028.424,E2 -18028.424} C_VEL
LIN {X 0,Y 419.316,Z 352.639,A -85,B 0,C 180,E1 -18029.007,E2 -18029.007} C_VEL
LIN {X 0,Y 418.651,Z 351.454,A -85,B 0,C 180,E1 -18029.207,E2 -18029.207} C_VEL
LIN {X 0,Y 416.436,Z 349.315,A -85,B 0,C 180,E1 -18029.817,E2 -18029.817} C_VEL
LIN {X 0,Y 415.433,Z 346.845,A -85,B 0,C 180,E1 -18030.195,E2 -18030.195} C_VEL
LIN {X 0,Y 415.348,Z 346.304,A -85,B 0,C 180,E1 -18030.283,E2 -18030.283} C_VEL
LIN {X 0,Y 415.331,Z 346.302,A -85,B 0,C 180,E1 -18033.816,E2 -18033.816} C_VEL
LIN {X 0,Y 415.33,Z 346.302,A -85,B 0,C 180,E1 -18036.176,E2 -18036.176} C_VEL
LIN {X 0,Y 415.293,Z 346.302,A -85,B 0,C 180,E1 -18039.117,E2 -18039.117} C_VEL
LIN {X 0,Y 415.281,Z 346.304,A -85,B 0,C 180,E1 -18042.428,E2 -18042.428} C_VEL
LIN {X 0,Y 415.303,Z 346.311,A -85,B 0,C 180,E1 -18045.102,E2 -18045.102} C_VEL
LIN {X 0,Y 415.279,Z 346.31,A -85,B 0,C 180,E1 -18047.914,E2 -18047.914} C_VEL
LIN {X 0,Y 415.283,Z 346.311,A -85,B 0,C 180,E1 -18051.386,E2 -18051.386} C_VEL
LIN {X 0,Y 415.314,Z 346.45,A -85,B 0,C 180,E1 -18054.53,E2 -18054.53} C_VEL
LIN {X 0,Y 419.282,Z 361.703,A -85,B 0,C 180,E1 -18057.465,E2 -18057.465} C_VEL
LIN {X 0,Y 422.249,Z 374.48,A -85,B 0,C 180,E1 -18059.763,E2 -18059.763} C_VEL
LIN {X 0,Y 425.687,Z 384.996,A -85,B 0,C 180,E1 -18060.853,E2 -18060.853} C_VEL
LIN {X 0,Y 428.971,Z 407.582,A -85,B 0,C 180,E1 -18062.359,E2 -18062.359} C_VEL
LIN {X 0,Y 431.568,Z 426.849,A -85,B 0,C 180,E1 -18063.497,E2 -18063.497} C_VEL
LIN {X 0,Y 433.443,Z 444.068,A -85,B 0,C 180,E1 -18064.393,E2 -18064.393} C_VEL
LIN {X 0,Y 434.579,Z 458.902,A -85,B 0,C 180,E1 -18065.085,E2 -18065.085} C_VEL
LIN {X 0,Y 435.238,Z 479.148,A -85,B 0,C 180,E1 -18065.876,E2 -18065.876} C_VEL
LIN {X 0,Y 430.254,Z 550.807,A -85,B 0,C 180,E1 -18067.822,E2 -18067.822} C_VEL
LIN {X 0,Y 428.668,Z 566.42,A -85,B 0,C 180,E1 -18068.429,E2 -18068.429} C_VEL
LIN {X 0,Y 426.823,Z 579.48,A -85,B 0,C 180,E1 -18069.088,E2 -18069.088} C_VEL
LIN {X 0,Y 424.579,Z 593.603,A -85,B 0,C 180,E1 -18070.007,E2 -18070.007} C_VEL
LIN {X 0,Y 422.498,Z 606.436,A -85,B 0,C 180,E1 -18071.046,E2 -18071.046} C_VEL
LIN {X 0,Y 420.558,Z 617.904,A -85,B 0,C 180,E1 -18072.179,E2 -18072.179} C_VEL
LIN {X 0,Y 418.654,Z 628.801,A -85,B 0,C 180,E1 -18073.475,E2 -18073.475} C_VEL
LIN {X 0,Y 416.946,Z 638.791,A -85,B 0,C 180,E1 -18074.907,E2 -18074.907} C_VEL
LIN {X 0,Y 415.468,Z 649.915,A -85,B 0,C 180,E1 -18076.844,E2 -18076.844} C_VEL
LIN {X 0,Y 415.016,Z 654.353,A -85,B 0,C 180,E1 -18077.697,E2 -18077.697} C_VEL
LIN {X 0,Y 414.343,Z 665.389,A -85,B 0,C 180,E1 -18079.124,E2 -18079.124} C_VEL
LIN {X 0,Y 413.878,Z 675.664,A -85,B 0,C 180,E1 -18080.748,E2 -18080.748} C_VEL
LIN {X 0,Y 413.476,Z 684.413,A -85,B 0,C 180,E1 -18082.456,E2 -18082.456} C_VEL
LIN {X 0,Y 413.327,Z 691.355,A -85,B 0,C 180,E1 -18084.164,E2 -18084.164} C_VEL
LIN {X 0,Y 413.198,Z 696.115,A -85,B 0,C 180,E1 -18085.625,E2 -18085.625} C_VEL
LIN {X 0,Y 413.159,Z 699.82,A -85,B 0,C 180,E1 -18087.085,E2 -18087.085} C_VEL
LIN {X 0,Y 413.176,Z 701.799,A -85,B 0,C 180,E1 -18088.057,E2 -18088.057} C_VEL
LIN {X 0,Y 413.17,Z 703.376,A -85,B 0,C 180,E1 -18089.028,E2 -18089.028} C_VEL
LIN {X 0,Y 413.127,Z 705.344,A -85,B 0,C 180,E1 -18090.971,E2 -18090.971} C_VEL
LIN {X 0,Y 413.168,Z 705.767,A -85,B 0,C 180,E1 -18091.943,E2 -18091.943} C_VEL
LIN {X 0,Y 413.212,Z 705.517,A -85,B 0,C 180,E1 -18093.888,E2 -18093.888} C_VEL
LIN {X 0,Y 413.515,Z 703.812,A -85,B 0,C 180,E1 -18095.833,E2 -18095.833} C_VEL
LIN {X 0,Y 414.076,Z 700.645,A -85,B 0,C 180,E1 -18097.777,E2 -18097.777} C_VEL
LIN {X 0,Y 414.9,Z 695.933,A -85,B 0,C 180,E1 -18099.719,E2 -18099.719} C_VEL
LIN {X 0,Y 415.937,Z 691.262,A -85,B 0,C 180,E1 -18101.166,E2 -18101.166} C_VEL
LIN {X 0,Y 417.294,Z 684.429,A -85,B 0,C 180,E1 -18102.876,E2 -18102.876} C_VEL
LIN {X 0,Y 418.889,Z 676.227,A -85,B 0,C 180,E1 -18104.526,E2 -18104.526} C_VEL
LIN {X 0,Y 420.696,Z 667.532,A -85,B 0,C 180,E1 -18105.945,E2 -18105.945} C_VEL
LIN {X 0,Y 422.573,Z 657.187,A -85,B 0,C 180,E1 -18107.359,E2 -18107.359} C_VEL
LIN {X 0,Y 424.679,Z 645.713,A -85,B 0,C 180,E1 -18108.636,E2 -18108.636} C_VEL
LIN {X 0,Y 426.783,Z 633.192,A -85,B 0,C 180,E1 -18109.786,E2 -18109.786} C_VEL
LIN {X 0,Y 428.845,Z 619.195,A -85,B 0,C 180,E1 -18110.809,E2 -18110.809} C_VEL
LIN {X 0,Y 430.8,Z 604.475,A -85,B 0,C 180,E1 -18111.646,E2 -18111.646} C_VEL
LIN {X 0,Y 432.492,Z 589.442,A -85,B 0,C 180,E1 -18112.281,E2 -18112.281} C_VEL
LIN {X 0,Y 434.361,Z 565.629,A -85,B 0,C 180,E1 -18112.976,E2 -18112.976} C_VEL
LIN {X 0,Y 440.786,Z 485.062,A -85,B 0,C 180,E1 -18115.219,E2 -18115.219} C_VEL
LIN {X 0,Y 441.132,Z 477.376,A -85,B 0,C 180,E1 -18115.477,E2 -18115.477} C_VEL
LIN {X 0,Y 440.716,Z 462.954,A -85,B 0,C 180,E1 -18116.108,E2 -18116.108} C_VEL
LIN {X 0,Y 439.35,Z 443.639,A -85,B 0,C 180,E1 -18117.104,E2 -18117.104} C_VEL
LIN {X 0,Y 438.658,Z 437.022,A -85,B 0,C 180,E1 -18117.505,E2 -18117.505} C_VEL
LIN {X 0,Y 439.427,Z 419.098,A -85,B 0,C 180,E1 -18119.088,E2 -18119.088} C_VEL
LIN {X 0,Y 440.609,Z 401.179,A -85,B 0,C 180,E1 -18120.919,E2 -18120.919} C_VEL
LIN {X 0,Y 440.889,Z 395.382,A -85,B 0,C 180,E1 -18121.619,E2 -18121.619} C_VEL
LIN {X 0,Y 440.389,Z 388.684,A -85,B 0,C 180,E1 -18122.736,E2 -18122.736} C_VEL
LIN {X 0,Y 440.04,Z 386.766,A -85,B 0,C 180,E1 -18123.134,E2 -18123.134} C_VEL
LIN {X 0,Y 436.813,Z 381.22,A -85,B 0,C 180,E1 -18125.259,E2 -18125.259} C_VEL
LIN {X 0,Y 435.232,Z 378.741,A -85,B 0,C 180,E1 -18126.546,E2 -18126.546} C_VEL
LIN {X 0,Y 434.025,Z 376.741,A -85,B 0,C 180,E1 -18127.825,E2 -18127.825} C_VEL
LIN {X 0,Y 432.953,Z 375.487,A -85,B 0,C 180,E1 -18129.12,E2 -18129.12} C_VEL
LIN {X 0,Y 432.213,Z 374.671,A -85,B 0,C 180,E1 -18130.409,E2 -18130.409} C_VEL
LIN {X 0,Y 431.763,Z 374.29,A -85,B 0,C 180,E1 -18131.733,E2 -18131.733} C_VEL
LIN {X 0,Y 431.629,Z 374.344,A -85,B 0,C 180,E1 -18133.092,E2 -18133.092} C_VEL
LIN {X 0,Y 431.85,Z 374.866,A -85,B 0,C 180,E1 -18134.466,E2 -18134.466} C_VEL
LIN {X 0,Y 432.243,Z 376.021,A -85,B 0,C 180,E1 -18135.829,E2 -18135.829} C_VEL
LIN {X 0,Y 433.271,Z 379.025,A -85,B 0,C 180,E1 -18138.044,E2 -18138.044} C_VEL
LIN {X 0,Y 434.505,Z 382.487,A -85,B 0,C 180,E1 -18139.848,E2 -18139.848} C_VEL
LIN {X 0,Y 436.153,Z 387.641,A -85,B 0,C 180,E1 -18141.899,E2 -18141.899} C_VEL
LIN {X 0,Y 437.987,Z 394.117,A -85,B 0,C 180,E1 -18143.969,E2 -18143.969} C_VEL
LIN {X 0,Y 439.745,Z 402.413,A -85,B 0,C 180,E1 -18146.117,E2 -18146.117} C_VEL
LIN {X 0,Y 440.795,Z 409.102,A -85,B 0,C 180,E1 -18147.621,E2 -18147.621} C_VEL
LIN {X 0,Y 440.924,Z 410.794,A -85,B 0,C 180,E1 -18147.955,E2 -18147.955} C_VEL
LIN {X 0,Y 436.937,Z 431.975,A -85,B 0,C 180,E1 -18150.992,E2 -18150.992} C_VEL
LIN {X 0,Y 435.634,Z 440.154,A -85,B 0,C 180,E1 -18152.112,E2 -18152.112} C_VEL
LIN {X 0,Y 439.031,Z 459.716,A -85,B 0,C 180,E1 -18153.444,E2 -18153.444} C_VEL
LIN {X 0,Y 441.129,Z 476.419,A -85,B 0,C 180,E1 -18154.393,E2 -18154.393} C_VEL
LIN {X 0,Y 441.427,Z 481.562,A -85,B 0,C 180,E1 -18154.632,E2 -18154.632} C_VEL
LIN {X 0,Y 435.094,Z 561.861,A -85,B 0,C 180,E1 -18156.841,E2 -18156.841} C_VEL
LIN {X 0,Y 433.232,Z 585.306,A -85,B 0,C 180,E1 -18157.513,E2 -18157.513} C_VEL
LIN {X 0,Y 431.546,Z 600.579,A -85,B 0,C 180,E1 -18158.143,E2 -18158.143} C_VEL
LIN {X 0,Y 429.856,Z 613.775,A -85,B 0,C 180,E1 -18158.868,E2 -18158.868} C_VEL
LIN {X 0,Y 427.947,Z 626.868,A -85,B 0,C 180,E1 -18159.772,E2 -18159.772} C_VEL
LIN {X 0,Y 425.776,Z 640.113,A -85,B 0,C 180,E1 -18160.916,E2 -18160.916} C_VEL
LIN {X 0,Y 423.605,Z 652.159,A -85,B 0,C 180,E1 -18162.188,E2 -18162.188} C_VEL
LIN {X 0,Y 421.476,Z 663.033,A -85,B 0,C 180,E1 -18163.59,E2 -18163.59} C_VEL
LIN {X 0,Y 419.408,Z 673.418,A -85,B 0,C 180,E1 -18165.245,E2 -18165.245} C_VEL
LIN {X 0,Y 417.696,Z 681.904,A -85,B 0,C 180,E1 -18166.916,E2 -18166.916} C_VEL
LIN {X 0,Y 416.54,Z 687.868,A -85,B 0,C 180,E1 -18168.359,E2 -18168.359} C_VEL
LIN {X 0,Y 415.395,Z 692.813,A -85,B 0,C 180,E1 -18169.802,E2 -18169.802} C_VEL
LIN {X 0,Y 414.362,Z 697.905,A -85,B 0,C 180,E1 -18171.739,E2 -18171.739} C_VEL
LIN {X 0,Y 413.804,Z 700.699,A -85,B 0,C 180,E1 -18173.195,E2 -18173.195} C_VEL
LIN {X 0,Y 413.341,Z 703.106,A -85,B 0,C 180,E1 -18175.14,E2 -18175.14} C_VEL
LIN {X 0,Y 413.097,Z 704.079,A -85,B 0,C 180,E1 -18177.084,E2 -18177.084} C_VEL
LIN {X 0,Y 413.095,Z 704.024,A -85,B 0,C 180,E1 -18178.057,E2 -18178.057} C_VEL
LIN {X 0,Y 413.07,Z 702.827,A -85,B 0,C 180,E1 -18180,E2 -18180} C_VEL
LIN {X 0,Y 413.095,Z 700.127,A -85,B 0,C 180,E1 -18181.944,E2 -18181.944} C_VEL
LIN {X 0,Y 413.126,Z 695.829,A -85,B 0,C 180,E1 -18183.889,E2 -18183.889} C_VEL
LIN {X 0,Y 413.25,Z 691.527,A -85,B 0,C 180,E1 -18185.349,E2 -18185.349} C_VEL
LIN {X 0,Y 413.454,Z 685.135,A -85,B 0,C 180,E1 -18187.055,E2 -18187.055} C_VEL
LIN {X 0,Y 413.805,Z 677.105,A -85,B 0,C 180,E1 -18188.763,E2 -18188.763} C_VEL
LIN {X 0,Y 414.209,Z 668.688,A -85,B 0,C 180,E1 -18190.228,E2 -18190.228} C_VEL
LIN {X 0,Y 414.828,Z 658.568,A -85,B 0,C 180,E1 -18191.691,E2 -18191.691} C_VEL
LIN {X 0,Y 415.545,Z 647.329,A -85,B 0,C 180,E1 -18193.03,E2 -18193.03} C_VEL
LIN {X 0,Y 416.211,Z 634.837,A -85,B 0,C 180,E1 -18194.249,E2 -18194.249} C_VEL
LIN {X 0,Y 417.114,Z 621.083,A -85,B 0,C 180,E1 -18195.337,E2 -18195.337} C_VEL
LIN {X 0,Y 417.899,Z 607.624,A -85,B 0,C 180,E1 -18196.18,E2 -18196.18} C_VEL
LIN {X 0,Y 418.396,Z 594.575,A -85,B 0,C 180,E1 -18196.817,E2 -18196.817} C_VEL
LIN {X 0,Y 418.96,Z 579.308,A -85,B 0,C 180,E1 -18197.357,E2 -18197.357} C_VEL
LIN {X 0,Y 421.836,Z 471.816,A -85,B 0,C 180,E1 -18199.933,E2 -18199.933} C_VEL
LIN {X 0,Y 418.906,Z 439.608,A -85,B 0,C 180,E1 -18200.816,E2 -18200.816} C_VEL
LIN {X 0,Y 420.657,Z 412.087,A -85,B 0,C 180,E1 -18204.338,E2 -18204.338} C_VEL
LIN {X 0,Y 422.421,Z 386.158,A -85,B 0,C 180,E1 -18207.664,E2 -18207.664} C_VEL
LIN {X 0,Y 422.861,Z 380.407,A -85,B 0,C 180,E1 -18208.402,E2 -18208.402} C_VEL
LIN {X 0,Y 419.791,Z 365.856,A -85,B 0,C 180,E1 -18210.452,E2 -18210.452} C_VEL
LIN {X 0,Y 415.361,Z 346.307,A -85,B 0,C 180,E1 -18213.306,E2 -18213.306} C_VEL
LIN {X 0,Y 415.334,Z 346.304,A -85,B 0,C 180,E1 -18216.176,E2 -18216.176} C_VEL
LIN {X 0,Y 415.324,Z 346.311,A -85,B 0,C 180,E1 -18219.123,E2 -18219.123} C_VEL
LIN {X 0,Y 415.323,Z 346.305,A -85,B 0,C 180,E1 -18222.424,E2 -18222.424} C_VEL
LIN {X 0,Y 415.348,Z 346.306,A -85,B 0,C 180,E1 -18225.097,E2 -18225.097} C_VEL
LIN {X 0,Y 415.317,Z 346.305,A -85,B 0,C 180,E1 -18227.909,E2 -18227.909} C_VEL
LIN {X 0,Y 415.335,Z 346.304,A -85,B 0,C 180,E1 -18231.392,E2 -18231.392} C_VEL
LIN {X 0,Y 415.341,Z 346.305,A -85,B 0,C 180,E1 -18235.013,E2 -18235.013} C_VEL
LIN {X 0,Y 415.327,Z 346.305,A -85,B 0,C 180,E1 -18238.479,E2 -18238.479} C_VEL
LIN {X 0,Y 415.351,Z 346.302,A -85,B 0,C 180,E1 -18241.824,E2 -18241.824} C_VEL
LIN {X 0,Y 415.339,Z 346.304,A -85,B 0,C 180,E1 -18245.064,E2 -18245.064} C_VEL
LIN {X 0,Y 415.391,Z 346.303,A -85,B 0,C 180,E1 -18248.225,E2 -18248.225} C_VEL
LIN {X 0,Y 415.397,Z 346.298,A -85,B 0,C 180,E1 -18251.314,E2 -18251.314} C_VEL
LIN {X 0,Y 415.364,Z 346.304,A -85,B 0,C 180,E1 -18252.968,E2 -18252.968} C_VEL
LIN {X 0,Y 417.719,Z 352.524,A -85,B 0,C 180,E1 -18253.211,E2 -18253.211} C_VEL
LIN {X 0,Y 425.284,Z 371.756,A -85,B 0,C 180,E1 -18253.931,E2 -18253.931} C_VEL
LIN {X 0,Y 425.508,Z 375.235,A -85,B 0,C 180,E1 -18254.003,E2 -18254.003} C_VEL
LIN {X 0,Y 424.223,Z 452.232,A -85,B 0,C 180,E1 -18255.294,E2 -18255.294} C_VEL
LIN {X 0,Y 424.148,Z 469.699,A -85,B 0,C 180,E1 -18255.658,E2 -18255.658} C_VEL
LIN {X 0,Y 423.819,Z 483.633,A -85,B 0,C 180,E1 -18256.135,E2 -18256.135} C_VEL
LIN {X 0,Y 423.225,Z 497.144,A -85,B 0,C 180,E1 -18256.785,E2 -18256.785} C_VEL
LIN {X 0,Y 422.474,Z 509.328,A -85,B 0,C 180,E1 -18257.553,E2 -18257.553} C_VEL
LIN {X 0,Y 421.578,Z 522.449,A -85,B 0,C 180,E1 -18258.603,E2 -18258.603} C_VEL
LIN {X 0,Y 420.576,Z 534.456,A -85,B 0,C 180,E1 -18259.808,E2 -18259.808} C_VEL
LIN {X 0,Y 419.406,Z 545.146,A -85,B 0,C 180,E1 -18261.113,E2 -18261.113} C_VEL
LIN {X 0,Y 418.318,Z 554.77,A -85,B 0,C 180,E1 -18262.544,E2 -18262.544} C_VEL
LIN {X 0,Y 417.311,Z 562.772,A -85,B 0,C 180,E1 -18263.978,E2 -18263.978} C_VEL
LIN {X 0,Y 416.419,Z 570.426,A -85,B 0,C 180,E1 -18265.659,E2 -18265.659} C_VEL
LIN {X 0,Y 415.828,Z 575.788,A -85,B 0,C 180,E1 -18267.104,E2 -18267.104} C_VEL
LIN {X 0,Y 415.266,Z 581.423,A -85,B 0,C 180,E1 -18269.034,E2 -18269.034} C_VEL
LIN {X 0,Y 414.883,Z 585.542,A -85,B 0,C 180,E1 -18270.968,E2 -18270.968} C_VEL
LIN {X 0,Y 414.871,Z 587.062,A -85,B 0,C 180,E1 -18271.935,E2 -18271.935} C_VEL
LIN {X 0,Y 414.645,Z 589.14,A -85,B 0,C 180,E1 -18273.875,E2 -18273.875} C_VEL
LIN {X 0,Y 414.775,Z 589.898,A -85,B 0,C 180,E1 -18275.816,E2 -18275.816} C_VEL
LIN {X 0,Y 415.012,Z 589.373,A -85,B 0,C 180,E1 -18277.76,E2 -18277.76} C_VEL
LIN {X 0,Y 415.413,Z 587.536,A -85,B 0,C 180,E1 -18279.707,E2 -18279.707} C_VEL
LIN {X 0,Y 416.122,Z 584.31,A -85,B 0,C 180,E1 -18281.654,E2 -18281.654} C_VEL
LIN {X 0,Y 417.027,Z 579.612,A -85,B 0,C 180,E1 -18283.6,E2 -18283.6} C_VEL
LIN {X 0,Y 418.238,Z 573.284,A -85,B 0,C 180,E1 -18285.543,E2 -18285.543} C_VEL
LIN {X 0,Y 419.461,Z 566.212,A -85,B 0,C 180,E1 -18287.242,E2 -18287.242} C_VEL
LIN {X 0,Y 420.739,Z 558.766,A -85,B 0,C 180,E1 -18288.692,E2 -18288.692} C_VEL
LIN {X 0,Y 422.147,Z 549.796,A -85,B 0,C 180,E1 -18290.139,E2 -18290.139} C_VEL
LIN {X 0,Y 423.689,Z 538.886,A -85,B 0,C 180,E1 -18291.583,E2 -18291.583} C_VEL
LIN {X 0,Y 425.033,Z 527.566,A -85,B 0,C 180,E1 -18292.799,E2 -18292.799} C_VEL
LIN {X 0,Y 426.413,Z 515.285,A -85,B 0,C 180,E1 -18293.86,E2 -18293.86} C_VEL
LIN {X 0,Y 427.439,Z 503.233,A -85,B 0,C 180,E1 -18294.7,E2 -18294.7} C_VEL
LIN {X 0,Y 428.094,Z 491.539,A -85,B 0,C 180,E1 -18295.355,E2 -18295.355} C_VEL
LIN {X 0,Y 428.109,Z 491.23,A -85,B 0,C 180,E1 -18295.37,E2 -18295.37} C_VEL
LIN {X 0,Y 427.827,Z 485.712,A -85,B 0,C 180,E1 -18295.657,E2 -18295.657} C_VEL
LIN {X 0,Y 425.498,Z 476.807,A -85,B 0,C 180,E1 -18296.157,E2 -18296.157} C_VEL
LIN {X 0,Y 423.082,Z 467.76,A -85,B 0,C 180,E1 -18296.589,E2 -18296.589} C_VEL
LIN {X 0,Y 422.543,Z 462.028,A -85,B 0,C 180,E1 -18296.752,E2 -18296.752} C_VEL
LIN {X 0,Y 424.205,Z 381.445,A -85,B 0,C 180,E1 -18298.132,E2 -18298.132} C_VEL
LIN {X 0,Y 414.575,Z 360.466,A -85,B 0,C 180,E1 -18299.18,E2 -18299.18} C_VEL
LIN {X 0,Y 408.429,Z 347.989,A -85,B 0,C 180,E1 -18299.862,E2 -18299.862} C_VEL
LIN {X 0,Y 408.295,Z 347.185,A -85,B 0,C 180,E1 -18299.906,E2 -18299.906} C_VEL
LIN {X 0,Y 408.224,Z 347.192,A -85,B 0,C 180,E1 -18303.303,E2 -18303.303} C_VEL
LIN {X 0,Y 408.215,Z 347.194,A -85,B 0,C 180,E1 -18306.91,E2 -18306.91} C_VEL
LIN {X 0,Y 408.231,Z 347.192,A -85,B 0,C 180,E1 -18309.456,E2 -18309.456} C_VEL
LIN {X 0,Y 408.226,Z 347.193,A -85,B 0,C 180,E1 -18312.455,E2 -18312.455} C_VEL
LIN {X 0,Y 408.273,Z 347.182,A -85,B 0,C 180,E1 -18315.298,E2 -18315.298} C_VEL
LIN {X 0,Y 408.239,Z 347.188,A -85,B 0,C 180,E1 -18319.021,E2 -18319.021} C_VEL
LIN {X 0,Y 408.255,Z 347.16,A -85,B 0,C 180,E1 -18322.114,E2 -18322.114} C_VEL
LIN {X 0,Y 408.243,Z 347.174,A -85,B 0,C 180,E1 -18325.514,E2 -18325.514} C_VEL
LIN {X 0,Y 408.267,Z 347.177,A -85,B 0,C 180,E1 -18329.074,E2 -18329.074} C_VEL
LIN {X 0,Y 408.286,Z 347.18,A -85,B 0,C 180,E1 -18332.406,E2 -18332.406} C_VEL
LIN {X 0,Y 408.298,Z 347.181,A -85,B 0,C 180,E1 -18335.686,E2 -18335.686} C_VEL
LIN {X 0,Y 408.318,Z 347.171,A -85,B 0,C 180,E1 -18338.885,E2 -18338.885} C_VEL
LIN {X 0,Y 414.361,Z 368.756,A -85,B 0,C 180,E1 -18339.587,E2 -18339.587} C_VEL
LIN {X 0,Y 412.166,Z 464.556,A -85,B 0,C 180,E1 -18341.9,E2 -18341.9} C_VEL
LIN {X 0,Y 411.904,Z 480.518,A -85,B 0,C 180,E1 -18342.495,E2 -18342.495} C_VEL
LIN {X 0,Y 411.414,Z 495.06,A -85,B 0,C 180,E1 -18343.24,E2 -18343.24} C_VEL
LIN {X 0,Y 410.82,Z 509.007,A -85,B 0,C 180,E1 -18344.169,E2 -18344.169} C_VEL
LIN {X 0,Y 410.143,Z 522.438,A -85,B 0,C 180,E1 -18345.283,E2 -18345.283} C_VEL
LIN {X 0,Y 409.586,Z 534.638,A -85,B 0,C 180,E1 -18346.526,E2 -18346.526} C_VEL
LIN {X 0,Y 409.051,Z 546.06,A -85,B 0,C 180,E1 -18347.942,E2 -18347.942} C_VEL
LIN {X 0,Y 408.476,Z 555.705,A -85,B 0,C 180,E1 -18349.377,E2 -18349.377} C_VEL
LIN {X 0,Y 408.036,Z 564.043,A -85,B 0,C 180,E1 -18350.863,E2 -18350.863} C_VEL
LIN {X 0,Y 407.662,Z 572.065,A -85,B 0,C 180,E1 -18352.596,E2 -18352.596} C_VEL
LIN {X 0,Y 407.477,Z 577.644,A -85,B 0,C 180,E1 -18354.08,E2 -18354.08} C_VEL
LIN {X 0,Y 407.448,Z 582.356,A -85,B 0,C 180,E1 -18355.624,E2 -18355.624} C_VEL
LIN {X 0,Y 407.489,Z 585.788,A -85,B 0,C 180,E1 -18357.044,E2 -18357.044} C_VEL
LIN {X 0,Y 407.621,Z 589.24,A -85,B 0,C 180,E1 -18359.015,E2 -18359.015} C_VEL
LIN {X 0,Y 407.931,Z 591.245,A -85,B 0,C 180,E1 -18360.984,E2 -18360.984} C_VEL
LIN {X 0,Y 408.526,Z 591.76,A -85,B 0,C 180,E1 -18362.948,E2 -18362.948} C_VEL
LIN {X 0,Y 409.378,Z 590.834,A -85,B 0,C 180,E1 -18364.907,E2 -18364.907} C_VEL
LIN {X 0,Y 410.434,Z 588.477,A -85,B 0,C 180,E1 -18366.861,E2 -18366.861} C_VEL
LIN {X 0,Y 411.486,Z 585.709,A -85,B 0,C 180,E1 -18368.319,E2 -18368.319} C_VEL
LIN {X 0,Y 413.295,Z 580.567,A -85,B 0,C 180,E1 -18370.252,E2 -18370.252} C_VEL
LIN {X 0,Y 414.678,Z 575.591,A -85,B 0,C 180,E1 -18371.694,E2 -18371.694} C_VEL
LIN {X 0,Y 416.5,Z 568.414,A -85,B 0,C 180,E1 -18373.37,E2 -18373.37} C_VEL
LIN {X 0,Y 418.61,Z 559.423,A -85,B 0,C 180,E1 -18375.032,E2 -18375.032} C_VEL
LIN {X 0,Y 420.459,Z 550.066,A -85,B 0,C 180,E1 -18376.451,E2 -18376.451} C_VEL
LIN {X 0,Y 422.644,Z 538.644,A -85,B 0,C 180,E1 -18377.854,E2 -18377.854} C_VEL
LIN {X 0,Y 424.569,Z 527.019,A -85,B 0,C 180,E1 -18379.016,E2 -18379.016} C_VEL
LIN {X 0,Y 426.568,Z 512.635,A -85,B 0,C 180,E1 -18380.171,E2 -18380.171} C_VEL
LIN {X 0,Y 427.912,Z 499.579,A -85,B 0,C 180,E1 -18381.014,E2 -18381.014} C_VEL
LIN {X 0,Y 429.128,Z 484.282,A -85,B 0,C 180,E1 -18381.766,E2 -18381.766} C_VEL
LIN {X 0,Y 429.999,Z 467.81,A -85,B 0,C 180,E1 -18382.349,E2 -18382.349} C_VEL
LIN {X 0,Y 435.536,Z 396.161,A -85,B 0,C 180,E1 -18384.352,E2 -18384.352} C_VEL
LIN {X 0,Y 435.89,Z 391.327,A -85,B 0,C 180,E1 -18384.497,E2 -18384.497} C_VEL
LIN {X 0,Y 430.357,Z 380.748,A -85,B 0,C 180,E1 -18385.723,E2 -18385.723} C_VEL
LIN {X 0,Y 423.834,Z 369.929,A -85,B 0,C 180,E1 -18387.265,E2 -18387.265} C_VEL
LIN {X 0,Y 421.064,Z 365.807,A -85,B 0,C 180,E1 -18387.974,E2 -18387.974} C_VEL
LIN {X 0,Y 418.521,Z 361.965,A -85,B 0,C 180,E1 -18388.663,E2 -18388.663} C_VEL
LIN {X 0,Y 416.071,Z 358.514,A -85,B 0,C 180,E1 -18389.349,E2 -18389.349} C_VEL
LIN {X 0,Y 415.3,Z 357.377,A -85,B 0,C 180,E1 -18389.584,E2 -18389.584} C_VEL
LIN {X 0,Y 412.998,Z 354.646,A -85,B 0,C 180,E1 -18390.272,E2 -18390.272} C_VEL
LIN {X 0,Y 412.058,Z 352.572,A -85,B 0,C 180,E1 -18390.62,E2 -18390.62} C_VEL
LIN {X 0,Y 409.612,Z 350.523,A -85,B 0,C 180,E1 -18391.372,E2 -18391.372} C_VEL
LIN {X 0,Y 408.416,Z 347.967,A -85,B 0,C 180,E1 -18391.88,E2 -18391.88} C_VEL
LIN {X 0,Y 408.266,Z 347.184,A -85,B 0,C 180,E1 -18392.011,E2 -18392.011} C_VEL
LIN {X 0,Y 408.316,Z 347.178,A -85,B 0,C 180,E1 -18394.571,E2 -18394.571} C_VEL
LIN {X 0,Y 408.267,Z 347.179,A -85,B 0,C 180,E1 -18398.143,E2 -18398.143} C_VEL
LIN {X 0,Y 408.251,Z 347.18,A -85,B 0,C 180,E1 -18400.981,E2 -18400.981} C_VEL
LIN {X 0,Y 408.272,Z 347.182,A -85,B 0,C 180,E1 -18404.701,E2 -18404.701} C_VEL
LIN {X 0,Y 408.24,Z 347.187,A -85,B 0,C 180,E1 -18407.998,E2 -18407.998} C_VEL
LIN {X 0,Y 408.246,Z 347.188,A -85,B 0,C 180,E1 -18411.854,E2 -18411.854} C_VEL
LIN {X 0,Y 408.209,Z 347.24,A -85,B 0,C 180,E1 -18414.067,E2 -18414.067} C_VEL
LIN {X 0,Y 411.976,Z 361.527,A -85,B 0,C 180,E1 -18416.891,E2 -18416.891} C_VEL
LIN {X 0,Y 417.466,Z 377.205,A -85,B 0,C 180,E1 -18419.015,E2 -18419.015} C_VEL
LIN {X 0,Y 418.659,Z 380.615,A -85,B 0,C 180,E1 -18419.418,E2 -18419.418} C_VEL
LIN {X 0,Y 421.219,Z 388.899,A -85,B 0,C 180,E1 -18420.297,E2 -18420.297} C_VEL
LIN {X 0,Y 424.176,Z 410.5,A -85,B 0,C 180,E1 -18421.775,E2 -18421.775} C_VEL
LIN {X 0,Y 426.527,Z 429.373,A -85,B 0,C 180,E1 -18422.921,E2 -18422.921} C_VEL
LIN {X 0,Y 428.088,Z 445.291,A -85,B 0,C 180,E1 -18423.782,E2 -18423.782} C_VEL
LIN {X 0,Y 429.202,Z 459.912,A -85,B 0,C 180,E1 -18424.48,E2 -18424.48} C_VEL
LIN {X 0,Y 429.657,Z 480.65,A -85,B 0,C 180,E1 -18425.318,E2 -18425.318} C_VEL
LIN {X 0,Y 424.597,Z 549.205,A -85,B 0,C 180,E1 -18427.222,E2 -18427.222} C_VEL
LIN {X 0,Y 422.807,Z 565.331,A -85,B 0,C 180,E1 -18427.859,E2 -18427.859} C_VEL
LIN {X 0,Y 420.604,Z 580.239,A -85,B 0,C 180,E1 -18428.636,E2 -18428.636} C_VEL
LIN {X 0,Y 418.331,Z 593.897,A -85,B 0,C 180,E1 -18429.554,E2 -18429.554} C_VEL
LIN {X 0,Y 416.084,Z 606.693,A -85,B 0,C 180,E1 -18430.63,E2 -18430.63} C_VEL
LIN {X 0,Y 413.872,Z 618.807,A -85,B 0,C 180,E1 -18431.881,E2 -18431.881} C_VEL
LIN {X 0,Y 411.883,Z 629.386,A -85,B 0,C 180,E1 -18433.196,E2 -18433.196} C_VEL
LIN {X 0,Y 410.098,Z 639.099,A -85,B 0,C 180,E1 -18434.648,E2 -18434.648} C_VEL
LIN {X 0,Y 408.657,Z 648.523,A -85,B 0,C 180,E1 -18436.368,E2 -18436.368} C_VEL
LIN {X 0,Y 407.856,Z 655.228,A -85,B 0,C 180,E1 -18437.792,E2 -18437.792} C_VEL
LIN {X 0,Y 407.258,Z 665.088,A -85,B 0,C 180,E1 -18439.094,E2 -18439.094} C_VEL
LIN {X 0,Y 406.841,Z 674.493,A -85,B 0,C 180,E1 -18440.586,E2 -18440.586} C_VEL
LIN {X 0,Y 406.411,Z 683.443,A -85,B 0,C 180,E1 -18442.324,E2 -18442.324} C_VEL
LIN {X 0,Y 406.238,Z 690.623,A -85,B 0,C 180,E1 -18444.062,E2 -18444.062} C_VEL
LIN {X 0,Y 406.123,Z 695.495,A -85,B 0,C 180,E1 -18445.549,E2 -18445.549} C_VEL
LIN {X 0,Y 406.074,Z 699.352,A -85,B 0,C 180,E1 -18447.034,E2 -18447.034} C_VEL
LIN {X 0,Y 406.092,Z 701.398,A -85,B 0,C 180,E1 -18448.023,E2 -18448.023} C_VEL
LIN {X 0,Y 406.064,Z 704.313,A -85,B 0,C 180,E1 -18450,E2 -18450} C_VEL
LIN {X 0,Y 406.087,Z 705.711,A -85,B 0,C 180,E1 -18451.977,E2 -18451.977} C_VEL
LIN {X 0,Y 406.132,Z 705.605,A -85,B 0,C 180,E1 -18453.956,E2 -18453.956} C_VEL
LIN {X 0,Y 406.452,Z 704.046,A -85,B 0,C 180,E1 -18455.935,E2 -18455.935} C_VEL
LIN {X 0,Y 407.064,Z 701.026,A -85,B 0,C 180,E1 -18457.912,E2 -18457.912} C_VEL
LIN {X 0,Y 407.921,Z 696.491,A -85,B 0,C 180,E1 -18459.887,E2 -18459.887} C_VEL
LIN {X 0,Y 409.03,Z 691.969,A -85,B 0,C 180,E1 -18461.357,E2 -18461.357} C_VEL
LIN {X 0,Y 410.429,Z 685.407,A -85,B 0,C 180,E1 -18463.079,E2 -18463.079} C_VEL
LIN {X 0,Y 412.113,Z 677.376,A -85,B 0,C 180,E1 -18464.77,E2 -18464.77} C_VEL
LIN {X 0,Y 413.997,Z 668.959,A -85,B 0,C 180,E1 -18466.21,E2 -18466.21} C_VEL
LIN {X 0,Y 415.986,Z 658.947,A -85,B 0,C 180,E1 -18467.643,E2 -18467.643} C_VEL
LIN {X 0,Y 418.176,Z 647.872,A -85,B 0,C 180,E1 -18468.937,E2 -18468.937} C_VEL
LIN {X 0,Y 420.358,Z 635.776,A -85,B 0,C 180,E1 -18470.101,E2 -18470.101} C_VEL
LIN {X 0,Y 422.489,Z 622.588,A -85,B 0,C 180,E1 -18471.137,E2 -18471.137} C_VEL
LIN {X 0,Y 424.504,Z 608.875,A -85,B 0,C 180,E1 -18471.984,E2 -18471.984} C_VEL
LIN {X 0,Y 426.271,Z 594.825,A -85,B 0,C 180,E1 -18472.651,E2 -18472.651} C_VEL
LIN {X 0,Y 427.805,Z 579.707,A -85,B 0,C 180,E1 -18473.173,E2 -18473.173} C_VEL
LIN {X 0,Y 435.185,Z 491.006,A -85,B 0,C 180,E1 -18475.695,E2 -18475.695} C_VEL
LIN {X 0,Y 436.007,Z 479.401,A -85,B 0,C 180,E1 -18476.061,E2 -18476.061} C_VEL
LIN {X 0,Y 435.715,Z 465.05,A -85,B 0,C 180,E1 -18476.707,E2 -18476.707} C_VEL
LIN {X 0,Y 434.52,Z 445.839,A -85,B 0,C 180,E1 -18477.724,E2 -18477.724} C_VEL
LIN {X 0,Y 433.671,Z 437.427,A -85,B 0,C 180,E1 -18478.256,E2 -18478.256} C_VEL
LIN {X 0,Y 434.563,Z 422.938,A -85,B 0,C 180,E1 -18479.566,E2 -18479.566} C_VEL
LIN {X 0,Y 435.465,Z 410.108,A -85,B 0,C 180,E1 -18480.887,E2 -18480.887} C_VEL
LIN {X 0,Y 436.343,Z 401.536,A -85,B 0,C 180,E1 -18481.828,E2 -18481.828} C_VEL
LIN {X 0,Y 436.362,Z 398.254,A -85,B 0,C 180,E1 -18482.303,E2 -18482.303} C_VEL
LIN {X 0,Y 435.908,Z 392.533,A -85,B 0,C 180,E1 -18483.325,E2 -18483.325} C_VEL
LIN {X 0,Y 433.203,Z 387.544,A -85,B 0,C 180,E1 -18485.171,E2 -18485.171} C_VEL
LIN {X 0,Y 430.786,Z 383.764,A -85,B 0,C 180,E1 -18487.182,E2 -18487.182} C_VEL
LIN {X 0,Y 429.604,Z 382.066,A -85,B 0,C 180,E1 -18488.5,E2 -18488.5} C_VEL
LIN {X 0,Y 428.147,Z 380.451,A -85,B 0,C 180,E1 -18490.874,E2 -18490.874} C_VEL
LIN {X 0,Y 427.651,Z 380.327,A -85,B 0,C 180,E1 -18493.465,E2 -18493.465} C_VEL
LIN {X 0,Y 427.955,Z 381.3,A -85,B 0,C 180,E1 -18495.268,E2 -18495.268} C_VEL
LIN {X 0,Y 428.648,Z 383.725,A -85,B 0,C 180,E1 -18497.336,E2 -18497.336} C_VEL
LIN {X 0,Y 429.751,Z 387.086,A -85,B 0,C 180,E1 -18499.311,E2 -18499.311} C_VEL
LIN {X 0,Y 431.074,Z 391.556,A -85,B 0,C 180,E1 -18501.255,E2 -18501.255} C_VEL
LIN {X 0,Y 432.6,Z 397.105,A -85,B 0,C 180,E1 -18503.196,E2 -18503.196} C_VEL
LIN {X 0,Y 434.089,Z 404.131,A -85,B 0,C 180,E1 -18505.182,E2 -18505.182} C_VEL
LIN {X 0,Y 435.327,Z 412.249,A -85,B 0,C 180,E1 -18507.12,E2 -18507.12} C_VEL
LIN {X 0,Y 435.432,Z 415.016,A -85,B 0,C 180,E1 -18507.676,E2 -18507.676} C_VEL
LIN {X 0,Y 430.44,Z 439.884,A -85,B 0,C 180,E1 -18511.259,E2 -18511.259} C_VEL
LIN {X 0,Y 433.576,Z 458.45,A -85,B 0,C 180,E1 -18512.608,E2 -18512.608} C_VEL
LIN {X 0,Y 435.649,Z 474.685,A -85,B 0,C 180,E1 -18513.6,E2 -18513.6} C_VEL
LIN {X 0,Y 436.21,Z 483.13,A -85,B 0,C 180,E1 -18514.025,E2 -18514.025} C_VEL
LIN {X 0,Y 429.573,Z 561.853,A -85,B 0,C 180,E1 -18516.245,E2 -18516.245} C_VEL
LIN {X 0,Y 427.654,Z 584.932,A -85,B 0,C 180,E1 -18516.917,E2 -18516.917} C_VEL
LIN {X 0,Y 425.974,Z 599.55,A -85,B 0,C 180,E1 -18517.523,E2 -18517.523} C_VEL
LIN {X 0,Y 424.041,Z 613.819,A -85,B 0,C 180,E1 -18518.309,E2 -18518.309} C_VEL
LIN {X 0,Y 422.031,Z 626.842,A -85,B 0,C 180,E1 -18519.221,E2 -18519.221} C_VEL
LIN {X 0,Y 419.702,Z 640.038,A -85,B 0,C 180,E1 -18520.375,E2 -18520.375} C_VEL
LIN {X 0,Y 417.43,Z 652.065,A -85,B 0,C 180,E1 -18521.662,E2 -18521.662} C_VEL
LIN {X 0,Y 415.16,Z 662.928,A -85,B 0,C 180,E1 -18523.08,E2 -18523.08} C_VEL
LIN {X 0,Y 413.267,Z 671.977,A -85,B 0,C 180,E1 -18524.518,E2 -18524.518} C_VEL
LIN {X 0,Y 411.368,Z 680.688,A -85,B 0,C 180,E1 -18526.209,E2 -18526.209} C_VEL
LIN {X 0,Y 410.089,Z 686.867,A -85,B 0,C 180,E1 -18527.672,E2 -18527.672} C_VEL
LIN {X 0,Y 408.729,Z 692.017,A -85,B 0,C 180,E1 -18529.134,E2 -18529.134} C_VEL
LIN {X 0,Y 407.613,Z 697.305,A -85,B 0,C 180,E1 -18531.103,E2 -18531.103} C_VEL
LIN {X 0,Y 406.769,Z 701.036,A -85,B 0,C 180,E1 -18533.077,E2 -18533.077} C_VEL
LIN {X 0,Y 406.264,Z 703.303,A -85,B 0,C 180,E1 -18535.055,E2 -18535.055} C_VEL
LIN {X 0,Y 406.001,Z 704.132,A -85,B 0,C 180,E1 -18537.033,E2 -18537.033} C_VEL
LIN {X 0,Y 405.994,Z 704.007,A -85,B 0,C 180,E1 -18538.023,E2 -18538.023} C_VEL
LIN {X 0,Y 405.972,Z 702.637,A -85,B 0,C 180,E1 -18540,E2 -18540} C_VEL
LIN {X 0,Y 405.998,Z 699.761,A -85,B 0,C 180,E1 -18541.978,E2 -18541.978} C_VEL
LIN {X 0,Y 406.017,Z 696.615,A -85,B 0,C 180,E1 -18543.462,E2 -18543.462} C_VEL
LIN {X 0,Y 406.127,Z 692.465,A -85,B 0,C 180,E1 -18544.947,E2 -18544.947} C_VEL
LIN {X 0,Y 406.27,Z 687.286,A -85,B 0,C 180,E1 -18546.435,E2 -18546.435} C_VEL
LIN {X 0,Y 406.571,Z 679.815,A -85,B 0,C 180,E1 -18548.172,E2 -18548.172} C_VEL
LIN {X 0,Y 406.988,Z 671.962,A -85,B 0,C 180,E1 -18549.66,E2 -18549.66} C_VEL
LIN {X 0,Y 407.467,Z 661.975,A -85,B 0,C 180,E1 -18551.224,E2 -18551.224} C_VEL
LIN {X 0,Y 408.223,Z 650.991,A -85,B 0,C 180,E1 -18552.637,E2 -18552.637} C_VEL
LIN {X 0,Y 408.862,Z 639.34,A -85,B 0,C 180,E1 -18553.878,E2 -18553.878} C_VEL
LIN {X 0,Y 409.682,Z 626.641,A -85,B 0,C 180,E1 -18554.987,E2 -18554.987} C_VEL
LIN {X 0,Y 410.489,Z 613.555,A -85,B 0,C 180,E1 -18555.908,E2 -18555.908} C_VEL
LIN {X 0,Y 411.023,Z 600.208,A -85,B 0,C 180,E1 -18556.649,E2 -18556.649} C_VEL
LIN {X 0,Y 411.727,Z 584.727,A -85,B 0,C 180,E1 -18557.289,E2 -18557.289} C_VEL
LIN {X 0,Y 412.255,Z 567.041,A -85,B 0,C 180,E1 -18557.776,E2 -18557.776} C_VEL
LIN {X 0,Y 414.778,Z 471.852,A -85,B 0,C 180,E1 -18560.11,E2 -18560.11} C_VEL
LIN {X 0,Y 411.966,Z 440.276,A -85,B 0,C 180,E1 -18560.985,E2 -18560.985} C_VEL
LIN {X 0,Y 411.983,Z 439.307,A -85,B 0,C 180,E1 -18561.049,E2 -18561.049} C_VEL
LIN {X 0,Y 413.821,Z 410.603,A -85,B 0,C 180,E1 -18564.767,E2 -18564.767} C_VEL
LIN {X 0,Y 415.677,Z 384.498,A -85,B 0,C 180,E1 -18568.153,E2 -18568.153} C_VEL
LIN {X 0,Y 415.92,Z 381.624,A -85,B 0,C 180,E1 -18568.527,E2 -18568.527} C_VEL
LIN {X 0,Y 412.602,Z 366.053,A -85,B 0,C 180,E1 -18570.749,E2 -18570.749} C_VEL
LIN {X 0,Y 408.318,Z 347.184,A -85,B 0,C 180,E1 -18573.516,E2 -18573.516} C_VEL
LIN {X 0,Y 408.275,Z 347.187,A -85,B 0,C 180,E1 -18576.904,E2 -18576.904} C_VEL
LIN {X 0,Y 408.286,Z 347.183,A -85,B 0,C 180,E1 -18579.465,E2 -18579.465} C_VEL
LIN {X 0,Y 408.277,Z 347.183,A -85,B 0,C 180,E1 -18582.463,E2 -18582.463} C_VEL
LIN {X 0,Y 408.313,Z 347.179,A -85,B 0,C 180,E1 -18585.304,E2 -18585.304} C_VEL
LIN {X 0,Y 408.275,Z 347.183,A -85,B 0,C 180,E1 -18588.003,E2 -18588.003} C_VEL
LIN {X 0,Y 408.269,Z 347.186,A -85,B 0,C 180,E1 -18590.596,E2 -18590.596} C_VEL
LIN {X 0,Y 408.28,Z 347.18,A -85,B 0,C 180,E1 -18593.74,E2 -18593.74} C_VEL
LIN {X 0,Y 408.275,Z 347.185,A -85,B 0,C 180,E1 -18596.702,E2 -18596.702} C_VEL
LIN {X 0,Y 408.293,Z 347.182,A -85,B 0,C 180,E1 -18600.165,E2 -18600.165} C_VEL
LIN {X 0,Y 408.342,Z 347.175,A -85,B 0,C 180,E1 -18603.513,E2 -18603.513} C_VEL
LIN {X 0,Y 408.302,Z 347.182,A -85,B 0,C 180,E1 -18606.761,E2 -18606.761} C_VEL
LIN {X 0,Y 408.383,Z 347.174,A -85,B 0,C 180,E1 -18610.622,E2 -18610.622} C_VEL
LIN {X 0,Y 408.339,Z 347.182,A -85,B 0,C 180,E1 -18612.607,E2 -18612.607} C_VEL
LIN {X 0,Y 410.898,Z 353.873,A -85,B 0,C 180,E1 -18612.879,E2 -18612.879} C_VEL
LIN {X 0,Y 418.734,Z 373.572,A -85,B 0,C 180,E1 -18613.641,E2 -18613.641} C_VEL
LIN {X 0,Y 417.525,Z 455.935,A -85,B 0,C 180,E1 -18615.053,E2 -18615.053} C_VEL
LIN {X 0,Y 417.41,Z 471.232,A -85,B 0,C 180,E1 -18615.39,E2 -18615.39} C_VEL
LIN {X 0,Y 417.035,Z 485.659,A -85,B 0,C 180,E1 -18615.905,E2 -18615.905} C_VEL
LIN {X 0,Y 416.322,Z 499.835,A -85,B 0,C 180,E1 -18616.624,E2 -18616.624} C_VEL
LIN {X 0,Y 415.51,Z 512.412,A -85,B 0,C 180,E1 -18617.465,E2 -18617.465} C_VEL
LIN {X 0,Y 414.621,Z 525.114,A -85,B 0,C 180,E1 -18618.543,E2 -18618.543} C_VEL
LIN {X 0,Y 413.56,Z 536.712,A -85,B 0,C 180,E1 -18619.756,E2 -18619.756} C_VEL
LIN {X 0,Y 412.465,Z 546.28,A -85,B 0,C 180,E1 -18620.963,E2 -18620.963} C_VEL
LIN {X 0,Y 411.362,Z 555.841,A -85,B 0,C 180,E1 -18622.417,E2 -18622.417} C_VEL
LIN {X 0,Y 410.329,Z 563.79,A -85,B 0,C 180,E1 -18623.876,E2 -18623.876} C_VEL
LIN {X 0,Y 409.407,Z 571.399,A -85,B 0,C 180,E1 -18625.585,E2 -18625.585} C_VEL
LIN {X 0,Y 408.809,Z 576.719,A -85,B 0,C 180,E1 -18627.054,E2 -18627.054} C_VEL
LIN {X 0,Y 408.224,Z 582.318,A -85,B 0,C 180,E1 -18629.017,E2 -18629.017} C_VEL
LIN {X 0,Y 407.844,Z 586.4,A -85,B 0,C 180,E1 -18630.984,E2 -18630.984} C_VEL
LIN {X 0,Y 407.648,Z 589.095,A -85,B 0,C 180,E1 -18632.955,E2 -18632.955} C_VEL
LIN {X 0,Y 407.7,Z 590.466,A -85,B 0,C 180,E1 -18634.928,E2 -18634.928} C_VEL
LIN {X 0,Y 407.857,Z 590.553,A -85,B 0,C 180,E1 -18636.905,E2 -18636.905} C_VEL
LIN {X 0,Y 408.191,Z 589.338,A -85,B 0,C 180,E1 -18638.884,E2 -18638.884} C_VEL
LIN {X 0,Y 408.687,Z 586.785,A -85,B 0,C 180,E1 -18640.867,E2 -18640.867} C_VEL
LIN {X 0,Y 409.595,Z 582.797,A -85,B 0,C 180,E1 -18642.845,E2 -18642.845} C_VEL
LIN {X 0,Y 410.719,Z 577.266,A -85,B 0,C 180,E1 -18644.822,E2 -18644.822} C_VEL
LIN {X 0,Y 411.72,Z 571.989,A -85,B 0,C 180,E1 -18646.303,E2 -18646.303} C_VEL
LIN {X 0,Y 412.91,Z 565.601,A -85,B 0,C 180,E1 -18647.779,E2 -18647.779} C_VEL
LIN {X 0,Y 414.213,Z 557.891,A -85,B 0,C 180,E1 -18649.254,E2 -18649.254} C_VEL
LIN {X 0,Y 415.718,Z 548.548,A -85,B 0,C 180,E1 -18650.722,E2 -18650.722} C_VEL
LIN {X 0,Y 417.225,Z 538.161,A -85,B 0,C 180,E1 -18652.064,E2 -18652.064} C_VEL
LIN {X 0,Y 418.606,Z 527.036,A -85,B 0,C 180,E1 -18653.247,E2 -18653.247} C_VEL
LIN {X 0,Y 419.907,Z 515.39,A -85,B 0,C 180,E1 -18654.253,E2 -18654.253} C_VEL
LIN {X 0,Y 420.953,Z 503.166,A -85,B 0,C 180,E1 -18655.107,E2 -18655.107} C_VEL
LIN {X 0,Y 421.627,Z 491.529,A -85,B 0,C 180,E1 -18655.756,E2 -18655.756} C_VEL
LIN {X 0,Y 422.221,Z 477.876,A -85,B 0,C 180,E1 -18656.323,E2 -18656.323} C_VEL
LIN {X 0,Y 422.49,Z 464.085,A -85,B 0,C 180,E1 -18656.711,E2 -18656.711} C_VEL
LIN {X 0,Y 422.543,Z 462.028,A -85,B 0,C 180,E1 -18656.752,E2 -18656.752} C_VEL
LIN {X 0,Y 422.079,Z 456.248,A -85,B 0,C 180,E1 -18656.901,E2 -18656.901} C_VEL
LIN {X 0,Y 417.221,Z 437.63,A -85,B 0,C 180,E1 -18657.548,E2 -18657.548} C_VEL
LIN {X 0,Y 416.665,Z 431.837,A -85,B 0,C 180,E1 -18657.69,E2 -18657.69} C_VEL
LIN {X 0,Y 417.719,Z 383.199,A -85,B 0,C 180,E1 -18658.532,E2 -18658.532} C_VEL
LIN {X 0,Y 408.314,Z 362.755,A -85,B 0,C 180,E1 -18659.583,E2 -18659.583} C_VEL
LIN {X 0,Y 401.481,Z 349.138,A -85,B 0,C 180,E1 -18660.361,E2 -18660.361} C_VEL
LIN {X 0,Y 401.269,Z 348.061,A -85,B 0,C 180,E1 -18660.412,E2 -18660.412} C_VEL
LIN {X 0,Y 401.164,Z 348.072,A -85,B 0,C 180,E1 -18663.968,E2 -18663.968} C_VEL
LIN {X 0,Y 401.21,Z 348.066,A -85,B 0,C 180,E1 -18667.665,E2 -18667.665} C_VEL
LIN {X 0,Y 401.187,Z 348.071,A -85,B 0,C 180,E1 -18671.344,E2 -18671.344} C_VEL
LIN {X 0,Y 401.218,Z 348.064,A -85,B 0,C 180,E1 -18674.293,E2 -18674.293} C_VEL
LIN {X 0,Y 401.198,Z 348.067,A -85,B 0,C 180,E1 -18677.162,E2 -18677.162} C_VEL
LIN {X 0,Y 401.18,Z 348.067,A -85,B 0,C 180,E1 -18680.195,E2 -18680.195} C_VEL
LIN {X 0,Y 401.188,Z 348.03,A -85,B 0,C 180,E1 -18683.586,E2 -18683.586} C_VEL
LIN {X 0,Y 401.214,Z 348.062,A -85,B 0,C 180,E1 -18687.234,E2 -18687.234} C_VEL
LIN {X 0,Y 401.234,Z 348.058,A -85,B 0,C 180,E1 -18690.794,E2 -18690.794} C_VEL
LIN {X 0,Y 401.269,Z 348.048,A -85,B 0,C 180,E1 -18694.126,E2 -18694.126} C_VEL
LIN {X 0,Y 401.204,Z 348.063,A -85,B 0,C 180,E1 -18697.715,E2 -18697.715} C_VEL
LIN {X 0,Y 401.289,Z 348.09,A -85,B 0,C 180,E1 -18698.721,E2 -18698.721} C_VEL
LIN {X 0,Y 407.33,Z 369.95,A -85,B 0,C 180,E1 -18699.441,E2 -18699.441} C_VEL
LIN {X 0,Y 405.129,Z 465.25,A -85,B 0,C 180,E1 -18701.802,E2 -18701.802} C_VEL
LIN {X 0,Y 404.87,Z 480.953,A -85,B 0,C 180,E1 -18702.397,E2 -18702.397} C_VEL
LIN {X 0,Y 404.359,Z 495.21,A -85,B 0,C 180,E1 -18703.133,E2 -18703.133} C_VEL
LIN {X 0,Y 403.792,Z 508.453,A -85,B 0,C 180,E1 -18704.015,E2 -18704.015} C_VEL
LIN {X 0,Y 403.163,Z 520.711,A -85,B 0,C 180,E1 -18705.023,E2 -18705.023} C_VEL
LIN {X 0,Y 402.566,Z 533.332,A -85,B 0,C 180,E1 -18706.286,E2 -18706.286} C_VEL
LIN {X 0,Y 402.086,Z 544.27,A -85,B 0,C 180,E1 -18707.606,E2 -18707.606} C_VEL
LIN {X 0,Y 401.465,Z 555.098,A -85,B 0,C 180,E1 -18709.189,E2 -18709.189} C_VEL
LIN {X 0,Y 400.908,Z 564.982,A -85,B 0,C 180,E1 -18710.953,E2 -18710.953} C_VEL
LIN {X 0,Y 400.55,Z 573.003,A -85,B 0,C 180,E1 -18712.716,E2 -18712.716} C_VEL
LIN {X 0,Y 400.37,Z 579.39,A -85,B 0,C 180,E1 -18714.478,E2 -18714.478} C_VEL
LIN {X 0,Y 400.415,Z 585.018,A -85,B 0,C 180,E1 -18716.49,E2 -18716.49} C_VEL
LIN {X 0,Y 400.413,Z 588.188,A -85,B 0,C 180,E1 -18717.995,E2 -18717.995} C_VEL
LIN {X 0,Y 400.664,Z 591.081,A -85,B 0,C 180,E1 -18720,E2 -18720} C_VEL
LIN {X 0,Y 401.138,Z 592.538,A -85,B 0,C 180,E1 -18722.001,E2 -18722.001} C_VEL
LIN {X 0,Y 401.918,Z 592.539,A -85,B 0,C 180,E1 -18723.997,E2 -18723.997} C_VEL
LIN {X 0,Y 402.957,Z 591.067,A -85,B 0,C 180,E1 -18725.986,E2 -18725.986} C_VEL
LIN {X 0,Y 404.158,Z 588.165,A -85,B 0,C 180,E1 -18727.969,E2 -18727.969} C_VEL
LIN {X 0,Y 405.992,Z 583.671,A -85,B 0,C 180,E1 -18729.935,E2 -18729.935} C_VEL
LIN {X 0,Y 407.54,Z 579.01,A -85,B 0,C 180,E1 -18731.45,E2 -18731.45} C_VEL
LIN {X 0,Y 409.307,Z 572.68,A -85,B 0,C 180,E1 -18733.105,E2 -18733.105} C_VEL
LIN {X 0,Y 411.456,Z 564.507,A -85,B 0,C 180,E1 -18734.794,E2 -18734.794} C_VEL
LIN {X 0,Y 413.688,Z 554.427,A -85,B 0,C 180,E1 -18736.475,E2 -18736.475} C_VEL
LIN {X 0,Y 415.928,Z 543.791,A -85,B 0,C 180,E1 -18737.899,E2 -18737.899} C_VEL
LIN {X 0,Y 418.151,Z 531.831,A -85,B 0,C 180,E1 -18739.192,E2 -18739.192} C_VEL
LIN {X 0,Y 420.006,Z 519.995,A -85,B 0,C 180,E1 -18740.246,E2 -18740.246} C_VEL
LIN {X 0,Y 421.827,Z 505.571,A -85,B 0,C 180,E1 -18741.278,E2 -18741.278} C_VEL
LIN {X 0,Y 423.129,Z 491.888,A -85,B 0,C 180,E1 -18742.049,E2 -18742.049} C_VEL
LIN {X 0,Y 424.149,Z 477.89,A -85,B 0,C 180,E1 -18742.643,E2 -18742.643} C_VEL
LIN {X 0,Y 425.356,Z 457.47,A -85,B 0,C 180,E1 -18743.279,E2 -18743.279} C_VEL
LIN {X 0,Y 430.722,Z 394.309,A -85,B 0,C 180,E1 -18745.087,E2 -18745.087} C_VEL
LIN {X 0,Y 425.797,Z 384.868,A -85,B 0,C 180,E1 -18746.241,E2 -18746.241} C_VEL
LIN {X 0,Y 420.051,Z 375.173,A -85,B 0,C 180,E1 -18747.676,E2 -18747.676} C_VEL
LIN {X 0,Y 414.983,Z 367.481,A -85,B 0,C 180,E1 -18749.071,E2 -18749.071} C_VEL
LIN {X 0,Y 412.059,Z 363.249,A -85,B 0,C 180,E1 -18749.956,E2 -18749.956} C_VEL
LIN {X 0,Y 409.557,Z 359.87,A -85,B 0,C 180,E1 -18750.753,E2 -18750.753} C_VEL
LIN {X 0,Y 408.737,Z 358.593,A -85,B 0,C 180,E1 -18751.036,E2 -18751.036} C_VEL
LIN {X 0,Y 406.49,Z 356.107,A -85,B 0,C 180,E1 -18751.821,E2 -18751.821} C_VEL
LIN {X 0,Y 405.335,Z 353.655,A -85,B 0,C 180,E1 -18752.323,E2 -18752.323} C_VEL
LIN {X 0,Y 402.724,Z 351.609,A -85,B 0,C 180,E1 -18753.29,E2 -18753.29} C_VEL
LIN {X 0,Y 401.49,Z 349.241,A -85,B 0,C 180,E1 -18753.936,E2 -18753.936} C_VEL
LIN {X 0,Y 401.241,Z 348.058,A -85,B 0,C 180,E1 -18754.244,E2 -18754.244} C_VEL
LIN {X 0,Y 401.23,Z 348.056,A -85,B 0,C 180,E1 -18757.662,E2 -18757.662} C_VEL
LIN {X 0,Y 401.195,Z 348.062,A -85,B 0,C 180,E1 -18761.345,E2 -18761.345} C_VEL
LIN {X 0,Y 401.243,Z 348.055,A -85,B 0,C 180,E1 -18764.296,E2 -18764.296} C_VEL
LIN {X 0,Y 401.196,Z 348.069,A -85,B 0,C 180,E1 -18767.161,E2 -18767.161} C_VEL
LIN {X 0,Y 401.177,Z 348.069,A -85,B 0,C 180,E1 -18770.195,E2 -18770.195} C_VEL
LIN {X 0,Y 401.205,Z 348.254,A -85,B 0,C 180,E1 -18772.613,E2 -18772.613} C_VEL
LIN {X 0,Y 402.069,Z 350.726,A -85,B 0,C 180,E1 -18773.186,E2 -18773.186} C_VEL
LIN {X 0,Y 403.655,Z 352.919,A -85,B 0,C 180,E1 -18773.943,E2 -18773.943} C_VEL
LIN {X 0,Y 408.401,Z 366.457,A -85,B 0,C 180,E1 -18776.376,E2 -18776.376} C_VEL
LIN {X 0,Y 413.874,Z 382.599,A -85,B 0,C 180,E1 -18778.609,E2 -18778.609} C_VEL
LIN {X 0,Y 416.856,Z 392.381,A -85,B 0,C 180,E1 -18779.692,E2 -18779.692} C_VEL
LIN {X 0,Y 419.452,Z 413.242,A -85,B 0,C 180,E1 -18781.162,E2 -18781.162} C_VEL
LIN {X 0,Y 421.955,Z 435.765,A -85,B 0,C 180,E1 -18782.552,E2 -18782.552} C_VEL
LIN {X 0,Y 423.784,Z 457.977,A -85,B 0,C 180,E1 -18783.727,E2 -18783.727} C_VEL
LIN {X 0,Y 424.318,Z 480.446,A -85,B 0,C 180,E1 -18784.681,E2 -18784.681} C_VEL
LIN {X 0,Y 418.947,Z 548.821,A -85,B 0,C 180,E1 -18786.637,E2 -18786.637} C_VEL
LIN {X 0,Y 417.182,Z 563.523,A -85,B 0,C 180,E1 -18787.218,E2 -18787.218} C_VEL
LIN {X 0,Y 415.069,Z 577.5,A -85,B 0,C 180,E1 -18787.946,E2 -18787.946} C_VEL
LIN {X 0,Y 412.381,Z 592.669,A -85,B 0,C 180,E1 -18788.972,E2 -18788.972} C_VEL
LIN {X 0,Y 409.864,Z 606.198,A -85,B 0,C 180,E1 -18790.12,E2 -18790.12} C_VEL
LIN {X 0,Y 407.369,Z 618.76,A -85,B 0,C 180,E1 -18791.452,E2 -18791.452} C_VEL
LIN {X 0,Y 405.126,Z 629.97,A -85,B 0,C 180,E1 -18792.907,E2 -18792.907} C_VEL
LIN {X 0,Y 403.266,Z 639.441,A -85,B 0,C 180,E1 -18794.382,E2 -18794.382} C_VEL
LIN {X 0,Y 401.736,Z 648.659,A -85,B 0,C 180,E1 -18796.129,E2 -18796.129} C_VEL
LIN {X 0,Y 400.672,Z 656.842,A -85,B 0,C 180,E1 -18797.997,E2 -18797.997} C_VEL
LIN {X 0,Y 400.165,Z 665.329,A -85,B 0,C 180,E1 -18799.154,E2 -18799.154} C_VEL
LIN {X 0,Y 399.726,Z 674.7,A -85,B 0,C 180,E1 -18800.672,E2 -18800.672} C_VEL
LIN {X 0,Y 399.334,Z 682.446,A -85,B 0,C 180,E1 -18802.187,E2 -18802.187} C_VEL
LIN {X 0,Y 399.164,Z 689.803,A -85,B 0,C 180,E1 -18803.956,E2 -18803.956} C_VEL
LIN {X 0,Y 399.063,Z 694.838,A -85,B 0,C 180,E1 -18805.47,E2 -18805.47} C_VEL
LIN {X 0,Y 398.996,Z 698.849,A -85,B 0,C 180,E1 -18806.981,E2 -18806.981} C_VEL
LIN {X 0,Y 398.998,Z 700.976,A -85,B 0,C 180,E1 -18807.988,E2 -18807.988} C_VEL
LIN {X 0,Y 398.995,Z 704.044,A -85,B 0,C 180,E1 -18810,E2 -18810} C_VEL
LIN {X 0,Y 398.985,Z 705.597,A -85,B 0,C 180,E1 -18812.012,E2 -18812.012} C_VEL
LIN {X 0,Y 399.048,Z 705.682,A -85,B 0,C 180,E1 -18814.026,E2 -18814.026} C_VEL
LIN {X 0,Y 399.402,Z 704.29,A -85,B 0,C 180,E1 -18816.04,E2 -18816.04} C_VEL
LIN {X 0,Y 400.039,Z 701.427,A -85,B 0,C 180,E1 -18818.052,E2 -18818.052} C_VEL
LIN {X 0,Y 400.948,Z 697.067,A -85,B 0,C 180,E1 -18820.061,E2 -18820.061} C_VEL
LIN {X 0,Y 402.131,Z 692.719,A -85,B 0,C 180,E1 -18821.555,E2 -18821.555} C_VEL
LIN {X 0,Y 403.863,Z 685.352,A -85,B 0,C 180,E1 -18823.545,E2 -18823.545} C_VEL
LIN {X 0,Y 405.346,Z 678.545,A -85,B 0,C 180,E1 -18825.023,E2 -18825.023} C_VEL
LIN {X 0,Y 407.313,Z 670.39,A -85,B 0,C 180,E1 -18826.484,E2 -18826.484} C_VEL
LIN {X 0,Y 409.42,Z 660.664,A -85,B 0,C 180,E1 -18827.936,E2 -18827.936} C_VEL
LIN {X 0,Y 411.903,Z 648.992,A -85,B 0,C 180,E1 -18829.366,E2 -18829.366} C_VEL
LIN {X 0,Y 414.175,Z 637.162,A -85,B 0,C 180,E1 -18830.544,E2 -18830.544} C_VEL
LIN {X 0,Y 416.4,Z 624.347,A -85,B 0,C 180,E1 -18831.59,E2 -18831.59} C_VEL
LIN {X 0,Y 418.642,Z 610.188,A -85,B 0,C 180,E1 -18832.503,E2 -18832.503} C_VEL
LIN {X 0,Y 420.475,Z 596.753,A -85,B 0,C 180,E1 -18833.176,E2 -18833.176} C_VEL
LIN {X 0,Y 422.238,Z 580.704,A -85,B 0,C 180,E1 -18833.757,E2 -18833.757} C_VEL
LIN {X 0,Y 430.238,Z 490.644,A -85,B 0,C 180,E1 -18836.38,E2 -18836.38} C_VEL
LIN {X 0,Y 430.992,Z 480.419,A -85,B 0,C 180,E1 -18836.715,E2 -18836.715} C_VEL
LIN {X 0,Y 430.798,Z 466.187,A -85,B 0,C 180,E1 -18837.376,E2 -18837.376} C_VEL
LIN {X 0,Y 429.851,Z 448.121,A -85,B 0,C 180,E1 -18838.366,E2 -18838.366} C_VEL
LIN {X 0,Y 428.916,Z 436.862,A -85,B 0,C 180,E1 -18839.112,E2 -18839.112} C_VEL
LIN {X 0,Y 429.922,Z 423.959,A -85,B 0,C 180,E1 -18840.335,E2 -18840.335} C_VEL
LIN {X 0,Y 431.742,Z 406.62,A -85,B 0,C 180,E1 -18842.208,E2 -18842.208} C_VEL
LIN {X 0,Y 432.014,Z 404.03,A -85,B 0,C 180,E1 -18842.531,E2 -18842.531} C_VEL
LIN {X 0,Y 431.797,Z 398.532,A -85,B 0,C 180,E1 -18843.472,E2 -18843.472} C_VEL
LIN {X 0,Y 431.109,Z 396.584,A -85,B 0,C 180,E1 -18844.043,E2 -18844.043} C_VEL
LIN {X 0,Y 429.262,Z 393.334,A -85,B 0,C 180,E1 -18845.327,E2 -18845.327} C_VEL
LIN {X 0,Y 426.835,Z 389.511,A -85,B 0,C 180,E1 -18847.386,E2 -18847.386} C_VEL
LIN {X 0,Y 425.197,Z 387.369,A -85,B 0,C 180,E1 -18849.263,E2 -18849.263} C_VEL
LIN {X 0,Y 424.084,Z 386.269,A -85,B 0,C 180,E1 -18851.351,E2 -18851.351} C_VEL
LIN {X 0,Y 423.709,Z 386.365,A -85,B 0,C 180,E1 -18853.972,E2 -18853.972} C_VEL
LIN {X 0,Y 424.049,Z 387.922,A -85,B 0,C 180,E1 -18856.072,E2 -18856.072} C_VEL
LIN {X 0,Y 424.712,Z 390.321,A -85,B 0,C 180,E1 -18857.915,E2 -18857.915} C_VEL
LIN {X 0,Y 425.833,Z 394.456,A -85,B 0,C 180,E1 -18860.096,E2 -18860.096} C_VEL
LIN {X 0,Y 427.283,Z 400.043,A -85,B 0,C 180,E1 -18862.314,E2 -18862.314} C_VEL
LIN {X 0,Y 428.656,Z 406.558,A -85,B 0,C 180,E1 -18864.347,E2 -18864.347} C_VEL
LIN {X 0,Y 429.809,Z 414.378,A -85,B 0,C 180,E1 -18866.352,E2 -18866.352} C_VEL
LIN {X 0,Y 430.112,Z 418.339,A -85,B 0,C 180,E1 -18867.227,E2 -18867.227} C_VEL
LIN {X 0,Y 425.505,Z 439.881,A -85,B 0,C 180,E1 -18870.39,E2 -18870.39} C_VEL
LIN {X 0,Y 428.122,Z 456.312,A -85,B 0,C 180,E1 -18871.657,E2 -18871.657} C_VEL
LIN {X 0,Y 430.202,Z 471.937,A -85,B 0,C 180,E1 -18872.701,E2 -18872.701} C_VEL
LIN {X 0,Y 431.191,Z 483.997,A -85,B 0,C 180,E1 -18873.374,E2 -18873.374} C_VEL
LIN {X 0,Y 424.214,Z 561.736,A -85,B 0,C 180,E1 -18875.62,E2 -18875.62} C_VEL
LIN {X 0,Y 422.183,Z 584.874,A -85,B 0,C 180,E1 -18876.309,E2 -18876.309} C_VEL
LIN {X 0,Y 420.309,Z 599.968,A -85,B 0,C 180,E1 -18876.944,E2 -18876.944} C_VEL
LIN {X 0,Y 418.301,Z 614.08,A -85,B 0,C 180,E1 -18877.737,E2 -18877.737} C_VEL
LIN {X 0,Y 416.193,Z 626.963,A -85,B 0,C 180,E1 -18878.658,E2 -18878.658} C_VEL
LIN {X 0,Y 413.717,Z 640.114,A -85,B 0,C 180,E1 -18879.821,E2 -18879.821} C_VEL
LIN {X 0,Y 411.304,Z 652.079,A -85,B 0,C 180,E1 -18881.121,E2 -18881.121} C_VEL
LIN {X 0,Y 408.92,Z 662.922,A -85,B 0,C 180,E1 -18882.557,E2 -18882.557} C_VEL
LIN {X 0,Y 406.897,Z 671.943,A -85,B 0,C 180,E1 -18884.013,E2 -18884.013} C_VEL
LIN {X 0,Y 404.794,Z 680.554,A -85,B 0,C 180,E1 -18885.699,E2 -18885.699} C_VEL
LIN {X 0,Y 403.217,Z 687.738,A -85,B 0,C 180,E1 -18887.459,E2 -18887.459} C_VEL
LIN {X 0,Y 401.807,Z 692.713,A -85,B 0,C 180,E1 -18888.945,E2 -18888.945} C_VEL
LIN {X 0,Y 400.608,Z 697.822,A -85,B 0,C 180,E1 -18890.947,E2 -18890.947} C_VEL
LIN {X 0,Y 399.744,Z 701.396,A -85,B 0,C 180,E1 -18892.955,E2 -18892.955} C_VEL
LIN {X 0,Y 399.202,Z 703.506,A -85,B 0,C 180,E1 -18894.967,E2 -18894.967} C_VEL
LIN {X 0,Y 398.928,Z 704.162,A -85,B 0,C 180,E1 -18896.981,E2 -18896.981} C_VEL
LIN {X 0,Y 398.856,Z 703.351,A -85,B 0,C 180,E1 -18898.994,E2 -18898.994} C_VEL
LIN {X 0,Y 398.891,Z 702.402,A -85,B 0,C 180,E1 -18900,E2 -18900} C_VEL
LIN {X 0,Y 398.925,Z 699.378,A -85,B 0,C 180,E1 -18902.013,E2 -18902.013} C_VEL
LIN {X 0,Y 398.987,Z 694.775,A -85,B 0,C 180,E1 -18904.027,E2 -18904.027} C_VEL
LIN {X 0,Y 399.1,Z 690.151,A -85,B 0,C 180,E1 -18905.54,E2 -18905.54} C_VEL
LIN {X 0,Y 399.35,Z 683.413,A -85,B 0,C 180,E1 -18907.306,E2 -18907.306} C_VEL
LIN {X 0,Y 399.713,Z 674.973,A -85,B 0,C 180,E1 -18909.074,E2 -18909.074} C_VEL
LIN {X 0,Y 400.209,Z 666.097,A -85,B 0,C 180,E1 -18910.59,E2 -18910.59} C_VEL
LIN {X 0,Y 400.849,Z 655.367,A -85,B 0,C 180,E1 -18912.104,E2 -18912.104} C_VEL
